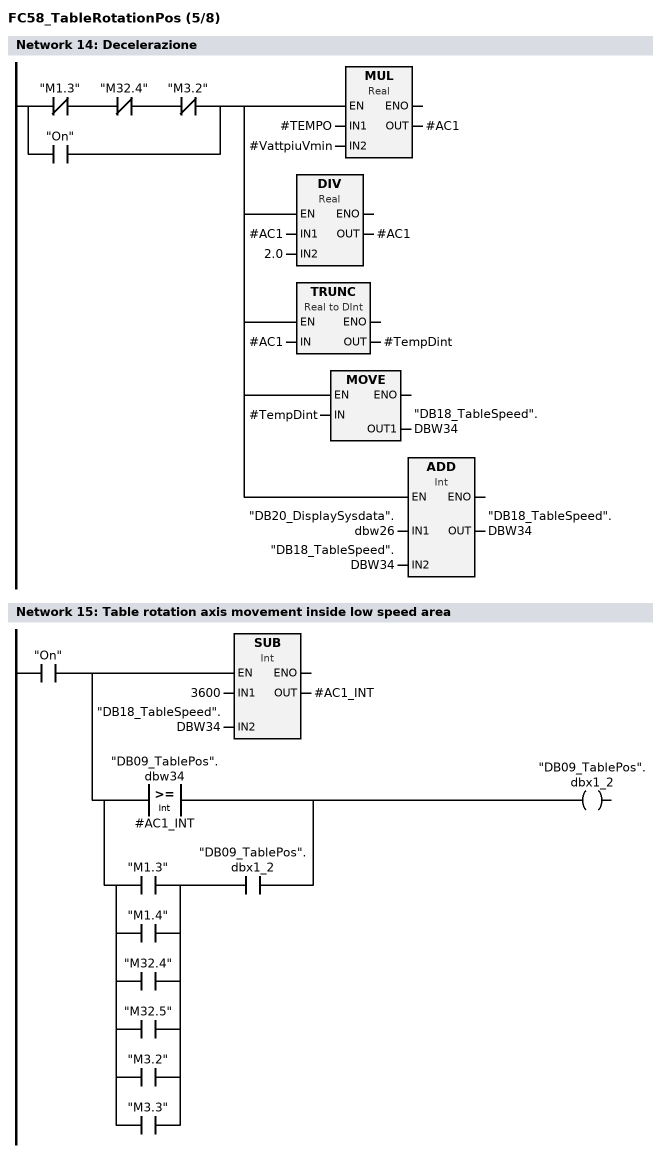
   RUNG wire#powerrail
      I_Contact( "M1.3" )
      I_Contact( "M32.4" )
      I_Contact( "M3.2" )
      wire#w1
      { S7_Templates := "SrcType := Real"; S7_GenerateENO := "TRUE" } Mul(in1 := #TEMPO, in2 := #VattpiuVmin, out => #AC1)
   END_RUNG
   RUNG wire#powerrail
      Contact( "On" )
   END_RUNG wire#w1
   RUNG wire#w1
      { S7_Templates := "SrcType := Real"; S7_GenerateENO := "TRUE" } Div(in1 := #AC1, in2 := 2.0, out => #AC1)
   END_RUNG
   RUNG wire#w1
      { S7_Templates := "[SrcType := Real, DestType := DInt]"; S7_GenerateENO := "TRUE" } Trunc(in := #AC1, out => #TempDint)
   END_RUNG
   RUNG wire#w1
      { S7_GenerateENO := "TRUE" } Move(in := #TempDint, out1 => "DB18_TableSpeed".DBW34)
   END_RUNG
   RUNG wire#w1
      { S7_Templates := "SrcType := Int"; S7_GenerateENO := "TRUE" } Add(in1 := "DB20_DisplaySysdata".dbw26, in2 := "DB18_TableSpeed".DBW34, out => "DB18_TableSpeed".DBW34)
   END_RUNG
   // the same network as SCL:
   IF (NOT "M1.3" AND NOT "M32.4" AND NOT "M3.2") OR "On" THEN
       #AC1 := #TEMPO * #VattpiuVmin;
       #AC1 := #AC1 / 2.0;
       #TempDint := TRUNC(#AC1);
       "DB18_TableSpeed".DBW34 := #TempDint;
       "DB18_TableSpeed".DBW34 := "DB20_DisplaySysdata".dbw26 + "DB18_TableSpeed".DBW34;
   END_IF;
END_REGION

REGION Network 15: Table rotation axis movement inside low speed area
   RUNG wire#powerrail
      Contact( "On" )
      wire#w1
      { S7_Templates := "SrcType := Int"; S7_GenerateENO := "TRUE" } Sub(in1 := 3600, in2 := "DB18_TableSpeed".DBW34, out => #AC1_INT)
   END_RUNG
   RUNG wire#w1
      { S7_Templates := "SrcType := Int" } GE_Contact(in1 := "DB09_TablePos".dbw34, in2 := #AC1_INT)
      wire#w2
      Coil( "DB09_TablePos".dbx1_2 )
   END_RUNG
   RUNG wire#w1
      Contact( "M1.3" )
      wire#w3
      Contact( "DB09_TablePos".dbx1_2 )
   END_RUNG wire#w2
   RUNG wire#w1
      Contact( "M1.4" )
   END_RUNG wire#w3
   RUNG wire#w1
      Contact( "M32.4" )
   END_RUNG wire#w3
   RUNG wire#w1
      Contact( "M32.5" )
   END_RUNG wire#w3
   RUNG wire#w1
      Contact( "M3.2" )
   END_RUNG wire#w3
   RUNG wire#w1
      Contact( "M3.3" )
   END_RUNG wire#w3
   // the same network as SCL:
   IF "On" THEN #AC1_INT := 3600 - "DB18_TableSpeed".DBW34; END_IF;
   "DB09_TablePos".dbx1_2 := "On" AND (("DB09_TablePos".dbw34 >= #AC1_INT) OR (("M1.3" OR "M1.4" OR "M32.4" OR "M32.5" OR "M3.2" OR "M3.3") AND "DB09_TablePos".dbx1_2));
END_REGION

REGION Network 16: Table rotation position loading/Unloading
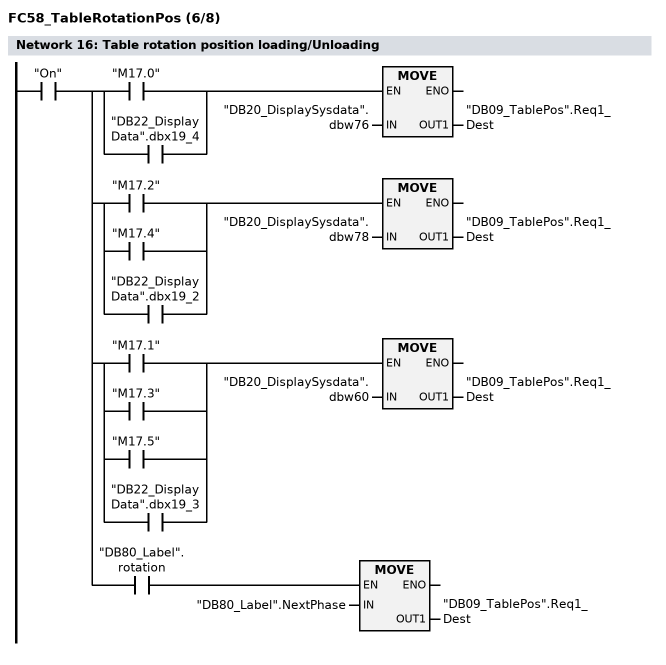
   RUNG wire#powerrail
      Contact( "On" )
      wire#w1
      Contact( "M17.0" )
      wire#w2
      { S7_GenerateENO := "TRUE" } Move(in := "DB20_DisplaySysdata".dbw76, out1 => "DB09_TablePos".Req1_Dest)
   END_RUNG
   RUNG wire#w1
      Contact( "DB22_DisplayData".dbx19_4 )
   END_RUNG wire#w2
   RUNG wire#w1
      Contact( "M17.2" )
      wire#w3
      { S7_GenerateENO := "TRUE" } Move(in := "DB20_DisplaySysdata".dbw78, out1 => "DB09_TablePos".Req1_Dest)
   END_RUNG
   RUNG wire#w1
      Contact( "M17.4" )
   END_RUNG wire#w3
   RUNG wire#w1
      Contact( "DB22_DisplayData".dbx19_2 )
   END_RUNG wire#w3
   RUNG wire#w1
      Contact( "M17.1" )
      wire#w4
      { S7_GenerateENO := "TRUE" } Move(in := "DB20_DisplaySysdata".dbw60, out1 => "DB09_TablePos".Req1_Dest)
   END_RUNG
   RUNG wire#w1
      Contact( "M17.3" )
   END_RUNG wire#w4
   RUNG wire#w1
      Contact( "M17.5" )
   END_RUNG wire#w4
   RUNG wire#w1
      Contact( "DB22_DisplayData".dbx19_3 )
   END_RUNG wire#w4
   RUNG wire#w1
      Contact( "DB80_Label".rotation )
      { S7_GenerateENO := "TRUE" } Move(in := "DB80_Label".NextPhase, out1 => "DB09_TablePos".Req1_Dest)
   END_RUNG
   // the same network as SCL:
   IF "On" AND ("M17.0" OR "DB22_DisplayData".dbx19_4) THEN
       "DB09_TablePos".Req1_Dest := "DB20_DisplaySysdata".dbw76;
   END_IF;
   IF "On" AND ("M17.2" OR "M17.4" OR "DB22_DisplayData".dbx19_2) THEN
       "DB09_TablePos".Req1_Dest := "DB20_DisplaySysdata".dbw78;
   END_IF;
   IF "On" AND ("M17.1" OR "M17.3" OR "M17.5" OR "DB22_DisplayData".dbx19_3) THEN
       "DB09_TablePos".Req1_Dest := "DB20_DisplaySysdata".dbw60;
   END_IF;
   IF "On" AND "DB80_Label".rotation THEN "DB09_TablePos".Req1_Dest := "DB80_Label".NextPhase; END_IF;
END_REGION

REGION Network 17
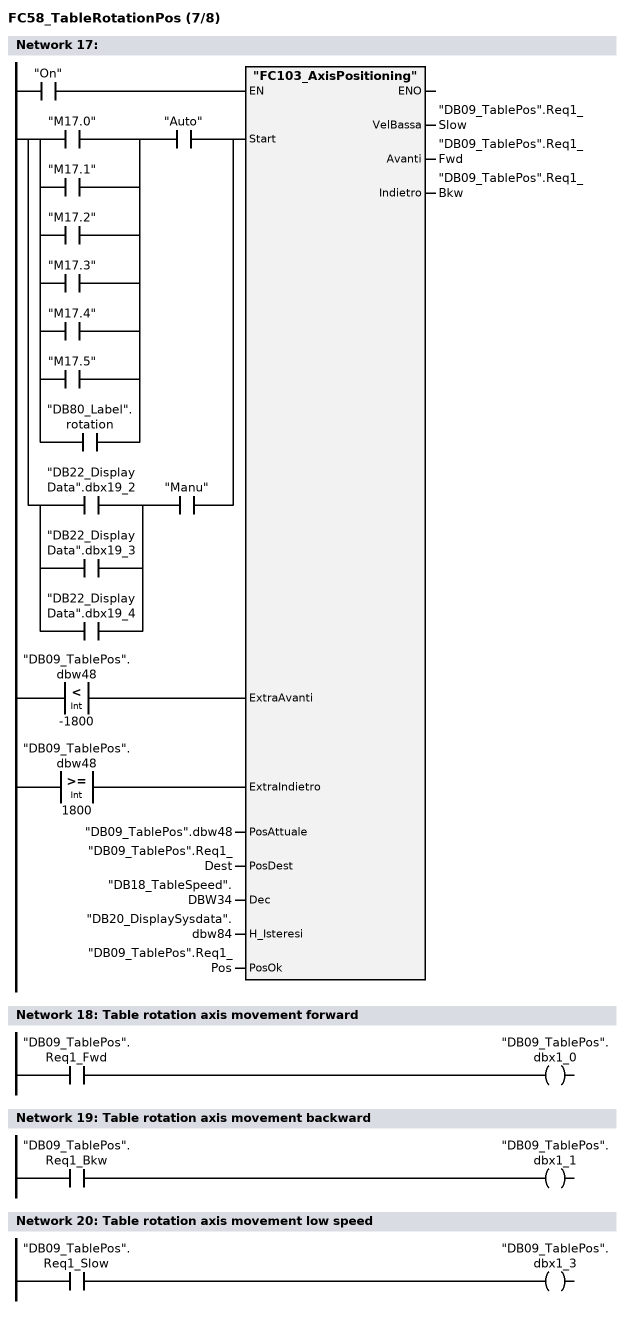
   RUNG wire#powerrail
      Contact( "On" )
      "FC103_AxisPositioning"(Start := wire#w3, ExtraAvanti := wire#w4, ExtraIndietro := wire#w5, PosAttuale := "DB09_TablePos".dbw48, PosDest := "DB09_TablePos".Req1_Dest, Dec := "DB18_TableSpeed".DBW34, H_Isteresi := "DB20_DisplaySysdata".dbw84, PosOk := "DB09_TablePos".Req1_Pos, VelBassa => "DB09_TablePos".Req1_Slow, Avanti => "DB09_TablePos".Req1_Fwd, Indietro => "DB09_TablePos".Req1_Bkw)
   END_RUNG
   RUNG wire#powerrail
      Contact( "M17.0" )
      wire#w1
      Contact( "Auto" )
   END_RUNG wire#w3
   RUNG wire#powerrail
      Contact( "M17.1" )
   END_RUNG wire#w1
   RUNG wire#powerrail
      Contact( "M17.2" )
   END_RUNG wire#w1
   RUNG wire#powerrail
      Contact( "M17.3" )
   END_RUNG wire#w1
   RUNG wire#powerrail
      Contact( "M17.4" )
   END_RUNG wire#w1
   RUNG wire#powerrail
      Contact( "M17.5" )
   END_RUNG wire#w1
   RUNG wire#powerrail
      Contact( "DB80_Label".rotation )
   END_RUNG wire#w1
   RUNG wire#powerrail
      Contact( "DB22_DisplayData".dbx19_2 )
      wire#w2
      Contact( "Manu" )
   END_RUNG wire#w3
   RUNG wire#powerrail
      Contact( "DB22_DisplayData".dbx19_3 )
   END_RUNG wire#w2
   RUNG wire#powerrail
      Contact( "DB22_DisplayData".dbx19_4 )
   END_RUNG wire#w2
   RUNG wire#powerrail
      { S7_Templates := "SrcType := Int" } LT_Contact(in1 := "DB09_TablePos".dbw48, in2 := -1800)
   END_RUNG wire#w4
   RUNG wire#powerrail
      { S7_Templates := "SrcType := Int" } GE_Contact(in1 := "DB09_TablePos".dbw48, in2 := 1800)
   END_RUNG wire#w5
   // the same network as SCL:
   IF "On" THEN
       "FC103_AxisPositioning"(Start := (("M17.0" OR "M17.1" OR "M17.2" OR "M17.3" OR "M17.4" OR "M17.5" OR "DB80_Label".rotation) AND "Auto") OR (("DB22_DisplayData".dbx19_2 OR "DB22_DisplayData".dbx19_3 OR "DB22_DisplayData".dbx19_4) AND "Manu"),
                               ExtraAvanti := "DB09_TablePos".dbw48 < (-1800),
                               ExtraIndietro := "DB09_TablePos".dbw48 >= 1800,
                               PosAttuale := "DB09_TablePos".dbw48,
                               PosDest := "DB09_TablePos".Req1_Dest,
                               Dec := "DB18_TableSpeed".DBW34,
                               H_Isteresi := "DB20_DisplaySysdata".dbw84,
                               PosOk := "DB09_TablePos".Req1_Pos,
                               VelBassa => "DB09_TablePos".Req1_Slow,
                               Avanti => "DB09_TablePos".Req1_Fwd,
                               Indietro => "DB09_TablePos".Req1_Bkw);
   END_IF;
END_REGION

REGION Network 18: Table rotation axis movement forward
   RUNG wire#powerrail
      Contact( "DB09_TablePos".Req1_Fwd )
      Coil( "DB09_TablePos".dbx1_0 )
   END_RUNG
   // the same network as SCL:
   "DB09_TablePos".dbx1_0 := "DB09_TablePos".Req1_Fwd;
END_REGION

REGION Network 19: Table rotation axis movement backward
   RUNG wire#powerrail
      Contact( "DB09_TablePos".Req1_Bkw )
      Coil( "DB09_TablePos".dbx1_1 )
   END_RUNG
   // the same network as SCL:
   "DB09_TablePos".dbx1_1 := "DB09_TablePos".Req1_Bkw;
END_REGION

REGION Network 20: Table rotation axis movement low speed
   RUNG wire#powerrail
      Contact( "DB09_TablePos".Req1_Slow )
      Coil( "DB09_TablePos".dbx1_3 )
   END_RUNG
   // the same network as SCL:
   "DB09_TablePos".dbx1_3 := "DB09_TablePos".Req1_Slow;
END_REGION

REGION Network 21: TABLE ENCODER CHECK
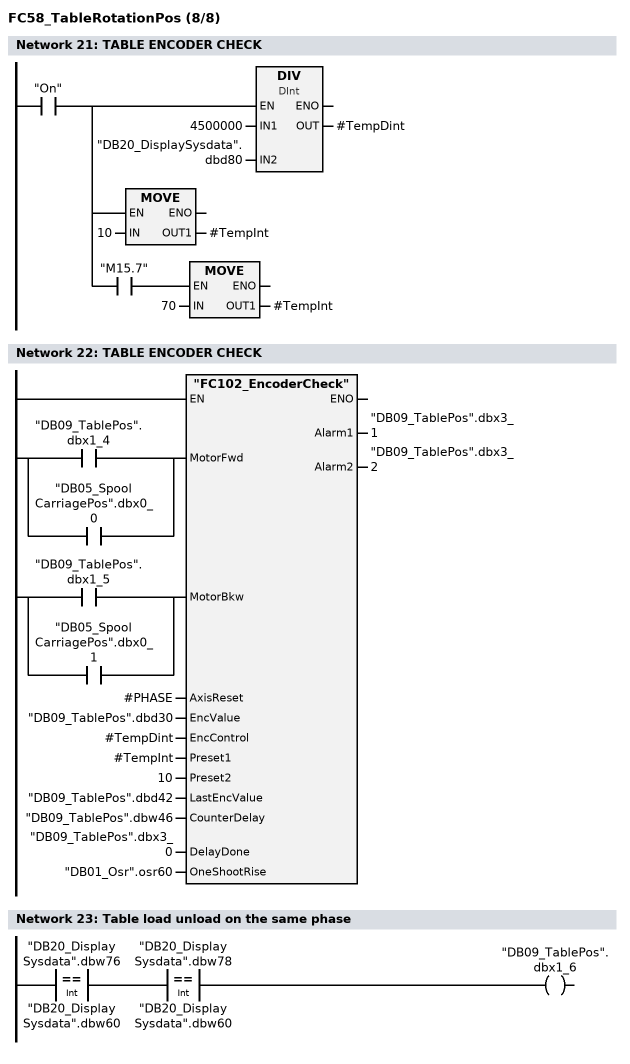
   RUNG wire#powerrail
      Contact( "On" )
      wire#w1
      { S7_Templates := "SrcType := DInt"; S7_GenerateENO := "TRUE" } Div(in1 := 4500000, in2 := "DB20_DisplaySysdata".dbd80, out => #TempDint)
   END_RUNG
   RUNG wire#w1
      { S7_GenerateENO := "TRUE" } Move(in := 10, out1 => #TempInt)
   END_RUNG
   RUNG wire#w1
      Contact( "M15.7" )
      { S7_GenerateENO := "TRUE" } Move(in := 70, out1 => #TempInt)
   END_RUNG
   // the same network as SCL:
   IF "On" THEN
       #TempDint := 4500000 / "DB20_DisplaySysdata".dbd80;
       #TempInt := 10;
   END_IF;
   IF "On" AND "M15.7" THEN #TempInt := 70; END_IF;
END_REGION

REGION Network 22: TABLE ENCODER CHECK
   RUNG wire#powerrail
      "FC102_EncoderCheck"(MotorFwd := wire#w1, MotorBkw := wire#w2, AxisReset := #PHASE, EncValue := "DB09_TablePos".dbd30, EncControl := #TempDint, Preset1 := #TempInt, Preset2 := 10, LastEncValue := "DB09_TablePos".dbd42, CounterDelay := "DB09_TablePos".dbw46, DelayDone := "DB09_TablePos".dbx3_0, OneShootRise := "DB01_Osr".osr60, Alarm1 => "DB09_TablePos".dbx3_1, Alarm2 => "DB09_TablePos".dbx3_2)
   END_RUNG
   RUNG wire#powerrail
      Contact( "DB09_TablePos".dbx1_4 )
   END_RUNG wire#w1
   RUNG wire#powerrail
      Contact( "DB05_SpoolCarriagePos".dbx0_0 )
   END_RUNG wire#w1
   RUNG wire#powerrail
      Contact( "DB09_TablePos".dbx1_5 )
   END_RUNG wire#w2
   RUNG wire#powerrail
      Contact( "DB05_SpoolCarriagePos".dbx0_1 )
   END_RUNG wire#w2
   // the same network as SCL:
   "FC102_EncoderCheck"(MotorFwd := "DB09_TablePos".dbx1_4 OR "DB05_SpoolCarriagePos".dbx0_0,
                        MotorBkw := "DB09_TablePos".dbx1_5 OR "DB05_SpoolCarriagePos".dbx0_1,
                        AxisReset := #PHASE,
                        EncValue := "DB09_TablePos".dbd30,
                        EncControl := #TempDint,
                        Preset1 := #TempInt,
                        Preset2 := 10,
                        LastEncValue := "DB09_TablePos".dbd42,
                        CounterDelay := "DB09_TablePos".dbw46,
                        DelayDone := "DB09_TablePos".dbx3_0,
                        OneShootRise := "DB01_Osr".osr60,
                        Alarm1 => "DB09_TablePos".dbx3_1,
                        Alarm2 => "DB09_TablePos".dbx3_2);
END_REGION

REGION Network 23: Table load unload on the same phase
   RUNG wire#powerrail
      { S7_Templates := "SrcType := Int" } EQ_Contact(in1 := "DB20_DisplaySysdata".dbw76, in2 := "DB20_DisplaySysdata".dbw60)
      { S7_Templates := "SrcType := Int" } EQ_Contact(in1 := "DB20_DisplaySysdata".dbw78, in2 := "DB20_DisplaySysdata".dbw60)
      Coil( "DB09_TablePos".dbx1_6 )
   END_RUNG
   // the same network as SCL:
   "DB09_TablePos".dbx1_6 := ("DB20_DisplaySysdata".dbw76 = "DB20_DisplaySysdata".dbw60) AND ("DB20_DisplaySysdata".dbw78 = "DB20_DisplaySysdata".dbw60);
END_REGION
END_FUNCTION

FUNCTION "FC62_PreStretchPGSAoutPWM" : Void   // FC62, LAD
{ S7_Optimized_Access := 'FALSE' }
AUTHOR : PaZan
VERSION : 0.1
// stored: AutoNumber false, IsIECCheckEnabled false, SetENOAutomatically false, UDAEnableTagReadback false
BEGIN

REGION Network 1: copy parameter for scale value % prestretch
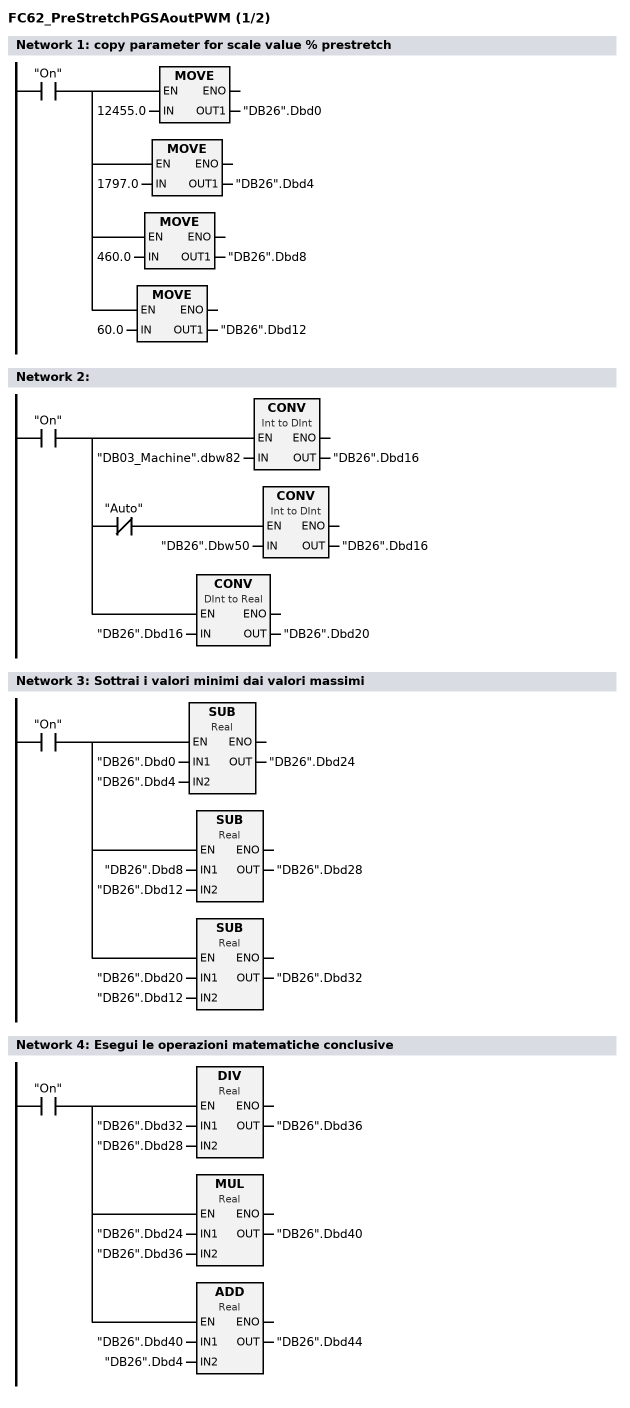
   RUNG wire#powerrail
      Contact( "On" )
      wire#w1
      { S7_GenerateENO := "TRUE" } Move(in := 12455.0, out1 => "DB26".Dbd0)
   END_RUNG
   RUNG wire#w1
      { S7_GenerateENO := "TRUE" } Move(in := 1797.0, out1 => "DB26".Dbd4)
   END_RUNG
   RUNG wire#w1
      { S7_GenerateENO := "TRUE" } Move(in := 460.0, out1 => "DB26".Dbd8)
   END_RUNG
   RUNG wire#w1
      { S7_GenerateENO := "TRUE" } Move(in := 60.0, out1 => "DB26".Dbd12)
   END_RUNG
   // the same network as SCL:
   IF "On" THEN
       "DB26".Dbd0 := 12455.0;
       "DB26".Dbd4 := 1797.0;
       "DB26".Dbd8 := 460.0;
       "DB26".Dbd12 := 60.0;
   END_IF;
END_REGION

REGION Network 2
   RUNG wire#powerrail
      Contact( "On" )
      wire#w1
      { S7_Templates := "[SrcType := Int, DestType := DInt]"; S7_GenerateENO := "TRUE" } Convert(in := "DB03_Machine".dbw82, out => "DB26".Dbd16)
   END_RUNG
   RUNG wire#w1
      I_Contact( "Auto" )
      { S7_Templates := "[SrcType := Int, DestType := DInt]"; S7_GenerateENO := "TRUE" } Convert(in := "DB26".Dbw50, out => "DB26".Dbd16)
   END_RUNG
   RUNG wire#w1
      { S7_Templates := "[SrcType := DInt, DestType := Real]"; S7_GenerateENO := "TRUE" } Convert(in := "DB26".Dbd16, out => "DB26".Dbd20)
   END_RUNG
   // the same network as SCL:
   IF "On" THEN "DB26".Dbd16 := INT_TO_DINT("DB03_Machine".dbw82); END_IF;
   IF "On" AND NOT "Auto" THEN "DB26".Dbd16 := INT_TO_DINT("DB26".Dbw50); END_IF;
   IF "On" THEN "DB26".Dbd20 := DINT_TO_REAL("DB26".Dbd16); END_IF;
END_REGION

REGION Network 3: Sottrai i valori minimi dai valori massimi
   RUNG wire#powerrail
      Contact( "On" )
      wire#w1
      { S7_Templates := "SrcType := Real"; S7_GenerateENO := "TRUE" } Sub(in1 := "DB26".Dbd0, in2 := "DB26".Dbd4, out => "DB26".Dbd24)
   END_RUNG
   RUNG wire#w1
      { S7_Templates := "SrcType := Real"; S7_GenerateENO := "TRUE" } Sub(in1 := "DB26".Dbd8, in2 := "DB26".Dbd12, out => "DB26".Dbd28)
   END_RUNG
   RUNG wire#w1
      { S7_Templates := "SrcType := Real"; S7_GenerateENO := "TRUE" } Sub(in1 := "DB26".Dbd20, in2 := "DB26".Dbd12, out => "DB26".Dbd32)
   END_RUNG
   // the same network as SCL:
   IF "On" THEN
       "DB26".Dbd24 := "DB26".Dbd0 - "DB26".Dbd4;
       "DB26".Dbd28 := "DB26".Dbd8 - "DB26".Dbd12;
       "DB26".Dbd32 := "DB26".Dbd20 - "DB26".Dbd12;
   END_IF;
END_REGION

REGION Network 4: Esegui le operazioni matematiche conclusive
   RUNG wire#powerrail
      Contact( "On" )
      wire#w1
      { S7_Templates := "SrcType := Real"; S7_GenerateENO := "TRUE" } Div(in1 := "DB26".Dbd32, in2 := "DB26".Dbd28, out => "DB26".Dbd36)
   END_RUNG
   RUNG wire#w1
      { S7_Templates := "SrcType := Real"; S7_GenerateENO := "TRUE" } Mul(in1 := "DB26".Dbd24, in2 := "DB26".Dbd36, out => "DB26".Dbd40)
   END_RUNG
   RUNG wire#w1
      { S7_Templates := "SrcType := Real"; S7_GenerateENO := "TRUE" } Add(in1 := "DB26".Dbd40, in2 := "DB26".Dbd4, out => "DB26".Dbd44)
   END_RUNG
   // the same network as SCL:
   IF "On" THEN
       "DB26".Dbd36 := "DB26".Dbd32 / "DB26".Dbd28;
       "DB26".Dbd40 := "DB26".Dbd24 * "DB26".Dbd36;
       "DB26".Dbd44 := "DB26".Dbd40 + "DB26".Dbd4;
   END_IF;
END_REGION

REGION Network 5: Trunc and copy value for pre-stretch in analogic out
   // PAW128
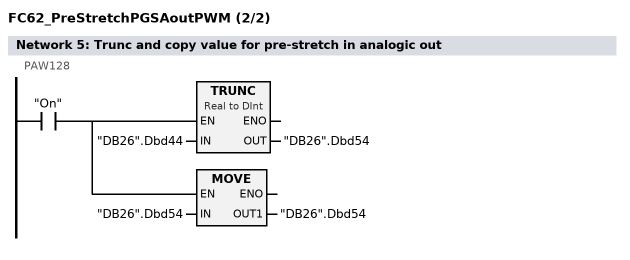
   RUNG wire#powerrail
      Contact( "On" )
      wire#w1
      { S7_Templates := "[SrcType := Real, DestType := DInt]"; S7_GenerateENO := "TRUE" } Trunc(in := "DB26".Dbd44, out => "DB26".Dbd54)
   END_RUNG
   RUNG wire#w1
      { S7_GenerateENO := "TRUE" } Move(in := "DB26".Dbd54, out1 => "DB26".Dbd54)
   END_RUNG
   // the same network as SCL:
   IF "On" THEN
       "DB26".Dbd54 := TRUNC("DB26".Dbd44);
       "DB26".Dbd54 := "DB26".Dbd54;
   END_IF;
END_REGION
END_FUNCTION

FUNCTION "FC71_Conveyor_0_IN_0_OUT" : Void   // FC71, LAD
TITLE = Conveyor_0_IN_0_OUT
{ S7_Optimized_Access := 'FALSE' }
VERSION : 0.1
// stored: AutoNumber false, IsIECCheckEnabled false, SetENOAutomatically false, UDAEnableTagReadback false
BEGIN

REGION Network 1: Conveyor manual movement
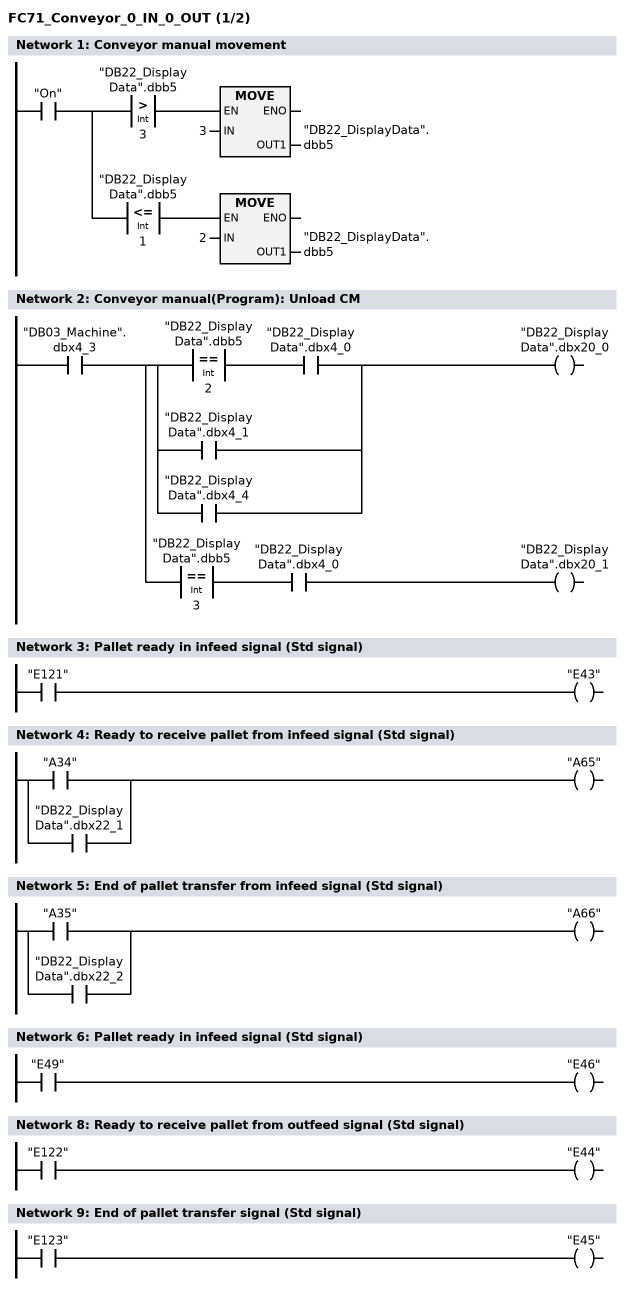
   RUNG wire#powerrail
      Contact( "On" )
      wire#w1
      { S7_Templates := "SrcType := Int" } GT_Contact(in1 := "DB22_DisplayData".dbb5, in2 := 3)
      { S7_GenerateENO := "TRUE" } Move(in := 3, out1 => "DB22_DisplayData".dbb5)
   END_RUNG
   RUNG wire#w1
      { S7_Templates := "SrcType := Int" } LE_Contact(in1 := "DB22_DisplayData".dbb5, in2 := 1)
      { S7_GenerateENO := "TRUE" } Move(in := 2, out1 => "DB22_DisplayData".dbb5)
   END_RUNG
   // the same network as SCL:
   IF "On" AND ("DB22_DisplayData".dbb5 > 3) THEN "DB22_DisplayData".dbb5 := 3; END_IF;
   IF "On" AND ("DB22_DisplayData".dbb5 <= 1) THEN "DB22_DisplayData".dbb5 := 2; END_IF;
END_REGION

REGION Network 2: Conveyor manual(Program): Unload CM
   RUNG wire#powerrail
      Contact( "DB03_Machine".dbx4_3 )
      wire#w1
      { S7_Templates := "SrcType := Int" } EQ_Contact(in1 := "DB22_DisplayData".dbb5, in2 := 2)
      Contact( "DB22_DisplayData".dbx4_0 )
      wire#w2
      Coil( "DB22_DisplayData".dbx20_0 )
   END_RUNG
   RUNG wire#w1
      Contact( "DB22_DisplayData".dbx4_1 )
   END_RUNG wire#w2
   RUNG wire#w1
      Contact( "DB22_DisplayData".dbx4_4 )
   END_RUNG wire#w2
   RUNG wire#w1
      { S7_Templates := "SrcType := Int" } EQ_Contact(in1 := "DB22_DisplayData".dbb5, in2 := 3)
      Contact( "DB22_DisplayData".dbx4_0 )
      Coil( "DB22_DisplayData".dbx20_1 )
   END_RUNG
   // the same network as SCL:
   "DB22_DisplayData".dbx20_0 := "DB03_Machine".dbx4_3 AND ((("DB22_DisplayData".dbb5 = 2) AND "DB22_DisplayData".dbx4_0) OR "DB22_DisplayData".dbx4_1 OR "DB22_DisplayData".dbx4_4);
   "DB22_DisplayData".dbx20_1 := "DB03_Machine".dbx4_3 AND ("DB22_DisplayData".dbb5 = 3) AND "DB22_DisplayData".dbx4_0;
END_REGION

REGION Network 3: Pallet ready in infeed signal (Std signal)
   RUNG wire#powerrail
      Contact( "E121" )
      Coil( "E43" )
   END_RUNG
   // the same network as SCL:
   "E43" := "E121";
END_REGION

REGION Network 4: Ready to receive pallet from infeed signal (Std signal)
   RUNG wire#powerrail
      Contact( "A34" )
      wire#w1
      Coil( "A65" )
   END_RUNG
   RUNG wire#powerrail
      Contact( "DB22_DisplayData".dbx22_1 )
   END_RUNG wire#w1
   // the same network as SCL:
   "A65" := "A34" OR "DB22_DisplayData".dbx22_1;
END_REGION

REGION Network 5: End of pallet transfer from infeed signal (Std signal)
   RUNG wire#powerrail
      Contact( "A35" )
      wire#w1
      Coil( "A66" )
   END_RUNG
   RUNG wire#powerrail
      Contact( "DB22_DisplayData".dbx22_2 )
   END_RUNG wire#w1
   // the same network as SCL:
   "A66" := "A35" OR "DB22_DisplayData".dbx22_2;
END_REGION

REGION Network 6: Pallet ready in infeed signal (Std signal)
   RUNG wire#powerrail
      Contact( "E49" )
      Coil( "E46" )
   END_RUNG
   // the same network as SCL:
   "E46" := "E49";
END_REGION

REGION Network 7: >>>>> OUTFEED CONVEYOR <<<<<<
END_REGION

REGION Network 8: Ready to receive pallet from outfeed signal (Std signal)
   RUNG wire#powerrail
      Contact( "E122" )
      Coil( "E44" )
   END_RUNG
   // the same network as SCL:
   "E44" := "E122";
END_REGION

REGION Network 9: End of pallet transfer signal (Std signal)
   RUNG wire#powerrail
      Contact( "E123" )
      Coil( "E45" )
   END_RUNG
   // the same network as SCL:
   "E45" := "E123";
END_REGION

REGION Network 10: Pallet ready for outfeed signal (Std signal)
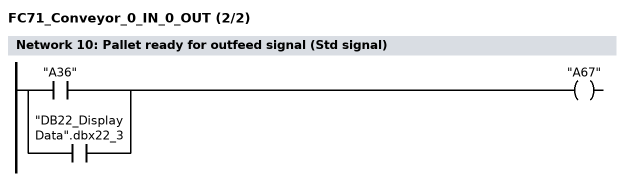
   RUNG wire#powerrail
      Contact( "A36" )
      wire#w1
      Coil( "A67" )
   END_RUNG
   RUNG wire#powerrail
      Contact( "DB22_DisplayData".dbx22_3 )
   END_RUNG wire#w1
   // the same network as SCL:
   "A67" := "A36" OR "DB22_DisplayData".dbx22_3;
END_REGION
END_FUNCTION

FUNCTION "FC72_Conveyor_0_IN_1_OUT" : Void   // FC72, LAD
TITLE = Conveyor_0_IN_1_OUT
{ S7_Optimized_Access := 'FALSE' }
VERSION : 0.1
// stored: AutoNumber false, IsIECCheckEnabled false, SetENOAutomatically false, UDAEnableTagReadback false
   VAR_TEMP   // added for the SCL form of the ladder/FBD networks
      _w1 : Bool;
   END_VAR
BEGIN

REGION Network 1: Conveyor manual movement
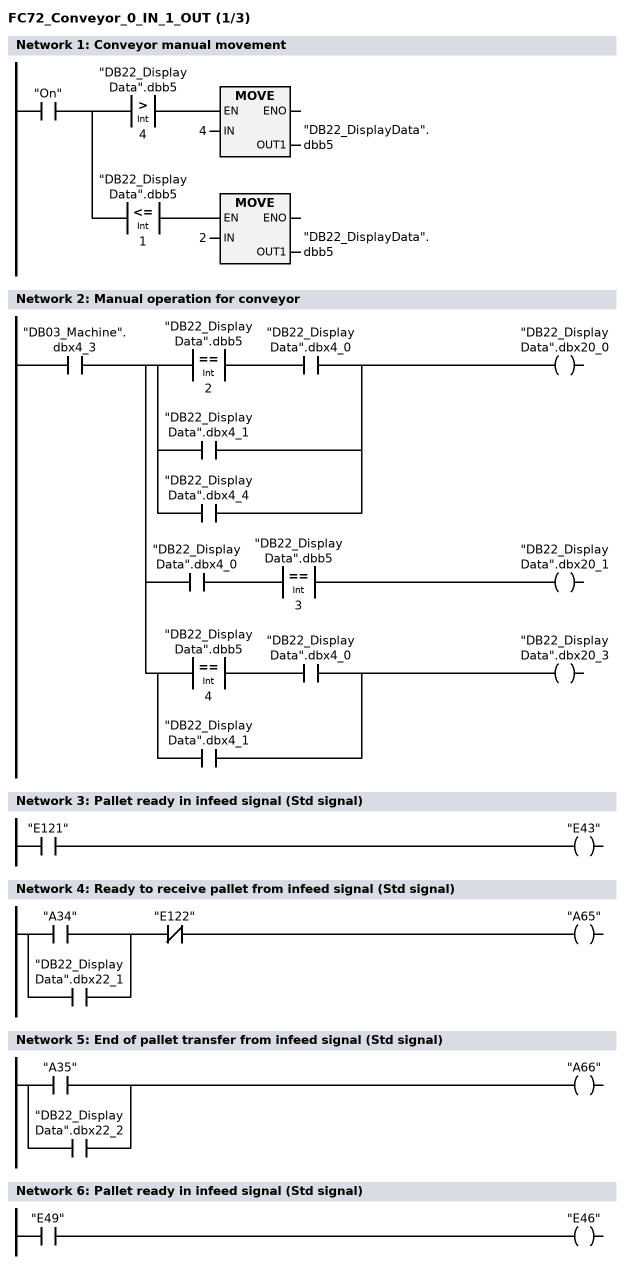
   RUNG wire#powerrail
      Contact( "On" )
      wire#w1
      { S7_Templates := "SrcType := Int" } GT_Contact(in1 := "DB22_DisplayData".dbb5, in2 := 4)
      { S7_GenerateENO := "TRUE" } Move(in := 4, out1 => "DB22_DisplayData".dbb5)
   END_RUNG
   RUNG wire#w1
      { S7_Templates := "SrcType := Int" } LE_Contact(in1 := "DB22_DisplayData".dbb5, in2 := 1)
      { S7_GenerateENO := "TRUE" } Move(in := 2, out1 => "DB22_DisplayData".dbb5)
   END_RUNG
   // the same network as SCL:
   IF "On" AND ("DB22_DisplayData".dbb5 > 4) THEN "DB22_DisplayData".dbb5 := 4; END_IF;
   IF "On" AND ("DB22_DisplayData".dbb5 <= 1) THEN "DB22_DisplayData".dbb5 := 2; END_IF;
END_REGION

REGION Network 2: Manual operation for conveyor
   RUNG wire#powerrail
      Contact( "DB03_Machine".dbx4_3 )
      wire#w1
      { S7_Templates := "SrcType := Int" } EQ_Contact(in1 := "DB22_DisplayData".dbb5, in2 := 2)
      Contact( "DB22_DisplayData".dbx4_0 )
      wire#w2
      Coil( "DB22_DisplayData".dbx20_0 )
   END_RUNG
   RUNG wire#w1
      Contact( "DB22_DisplayData".dbx4_1 )
   END_RUNG wire#w2
   RUNG wire#w1
      Contact( "DB22_DisplayData".dbx4_4 )
   END_RUNG wire#w2
   RUNG wire#w1
      Contact( "DB22_DisplayData".dbx4_0 )
      { S7_Templates := "SrcType := Int" } EQ_Contact(in1 := "DB22_DisplayData".dbb5, in2 := 3)
      Coil( "DB22_DisplayData".dbx20_1 )
   END_RUNG
   RUNG wire#w1
      { S7_Templates := "SrcType := Int" } EQ_Contact(in1 := "DB22_DisplayData".dbb5, in2 := 4)
      Contact( "DB22_DisplayData".dbx4_0 )
      wire#w3
      Coil( "DB22_DisplayData".dbx20_3 )
   END_RUNG
   RUNG wire#w1
      Contact( "DB22_DisplayData".dbx4_1 )
   END_RUNG wire#w3
   // the same network as SCL:
   "DB22_DisplayData".dbx20_0 := "DB03_Machine".dbx4_3 AND ((("DB22_DisplayData".dbb5 = 2) AND "DB22_DisplayData".dbx4_0) OR "DB22_DisplayData".dbx4_1 OR "DB22_DisplayData".dbx4_4);
   "DB22_DisplayData".dbx20_1 := "DB03_Machine".dbx4_3 AND "DB22_DisplayData".dbx4_0 AND ("DB22_DisplayData".dbb5 = 3);
   "DB22_DisplayData".dbx20_3 := "DB03_Machine".dbx4_3 AND ((("DB22_DisplayData".dbb5 = 4) AND "DB22_DisplayData".dbx4_0) OR "DB22_DisplayData".dbx4_1);
END_REGION

REGION Network 3: Pallet ready in infeed signal (Std signal)
   RUNG wire#powerrail
      Contact( "E121" )
      Coil( "E43" )
   END_RUNG
   // the same network as SCL:
   "E43" := "E121";
END_REGION

REGION Network 4: Ready to receive pallet from infeed signal (Std signal)
   RUNG wire#powerrail
      Contact( "A34" )
      wire#w1
      I_Contact( "E122" )
      Coil( "A65" )
   END_RUNG
   RUNG wire#powerrail
      Contact( "DB22_DisplayData".dbx22_1 )
   END_RUNG wire#w1
   // the same network as SCL:
   "A65" := ("A34" OR "DB22_DisplayData".dbx22_1) AND NOT "E122";
END_REGION

REGION Network 5: End of pallet transfer from infeed signal (Std signal)
   RUNG wire#powerrail
      Contact( "A35" )
      wire#w1
      Coil( "A66" )
   END_RUNG
   RUNG wire#powerrail
      Contact( "DB22_DisplayData".dbx22_2 )
   END_RUNG wire#w1
   // the same network as SCL:
   "A66" := "A35" OR "DB22_DisplayData".dbx22_2;
END_REGION

REGION Network 6: Pallet ready in infeed signal (Std signal)
   RUNG wire#powerrail
      Contact( "E49" )
      Coil( "E46" )
   END_RUNG
   // the same network as SCL:
   "E46" := "E49";
END_REGION

REGION Network 7: >>>>> OUTFEED CONVEYOR <<<<<<
END_REGION

REGION Network 8: Time for pallet unload with forklift
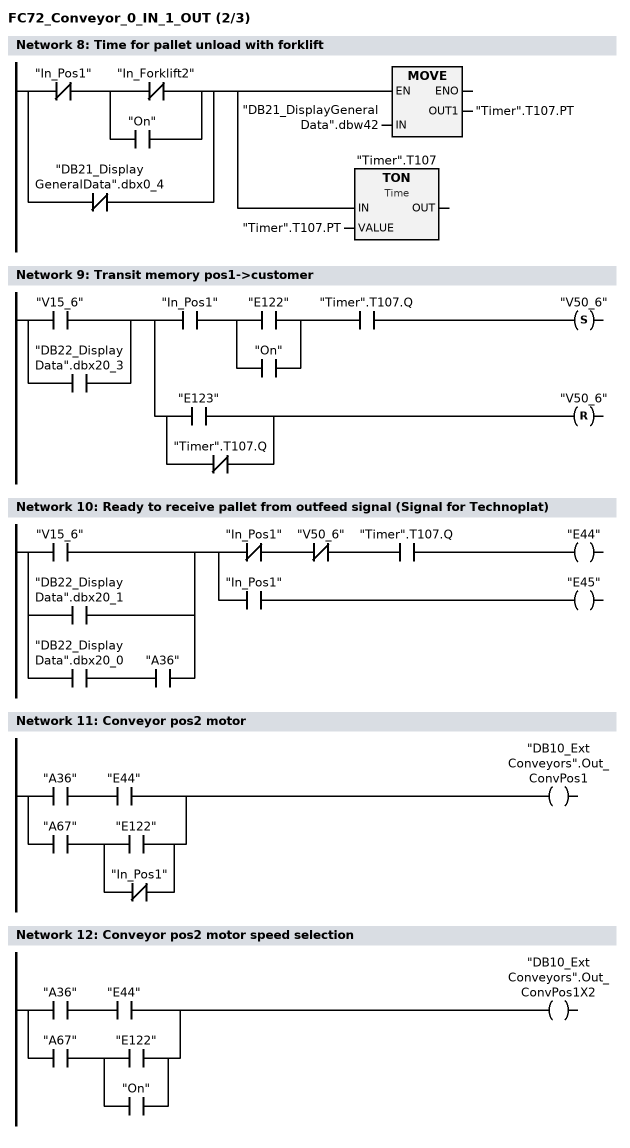
   #_w1 := (NOT "In_Pos1" AND (NOT "In_Forklift2" OR "On")) OR NOT "DB21_DisplayGeneralData".dbx0_4;
   IF #_w1 THEN "Timer".T107.PT := "DB21_DisplayGeneralData".dbw42; END_IF;
   "Timer".T107.TON(IN := #_w1, PT := "Timer".T107.PT);   // TON coil
END_REGION

REGION Network 9: Transit memory pos1->customer
   RUNG wire#powerrail
      Contact( "V15_6" )
      wire#w1
      Contact( "In_Pos1" )
      wire#w2
      Contact( "E122" )
      wire#w3
      Contact( "Timer".T107.Q )
      S_Coil( "V50_6" )
   END_RUNG
   RUNG wire#powerrail
      Contact( "DB22_DisplayData".dbx20_3 )
   END_RUNG wire#w1
   RUNG wire#w2
      Contact( "On" )
   END_RUNG wire#w3
   RUNG wire#w1
      Contact( "E123" )
      wire#w4
      R_Coil( "V50_6" )
   END_RUNG
   RUNG wire#w1
      I_Contact( "Timer".T107.Q )
   END_RUNG wire#w4
   // the same network as SCL:
   #_w1 := "V15_6" OR "DB22_DisplayData".dbx20_3;
   IF #_w1 AND "In_Pos1" AND ("E122" OR "On") AND "Timer".T107.Q THEN "V50_6" := TRUE; END_IF;
   IF #_w1 AND ("E123" OR NOT "Timer".T107.Q) THEN "V50_6" := FALSE; END_IF;
END_REGION

REGION Network 10: Ready to receive pallet from outfeed signal (Signal for Technoplat)
   RUNG wire#powerrail
      Contact( "V15_6" )
      wire#w1
      I_Contact( "In_Pos1" )
      I_Contact( "V50_6" )
      Contact( "Timer".T107.Q )
      Coil( "E44" )
   END_RUNG
   RUNG wire#powerrail
      Contact( "DB22_DisplayData".dbx20_1 )
   END_RUNG wire#w1
   RUNG wire#powerrail
      Contact( "DB22_DisplayData".dbx20_0 )
      Contact( "A36" )
   END_RUNG wire#w1
   RUNG wire#w1
      Contact( "In_Pos1" )
      Coil( "E45" )
   END_RUNG
   // the same network as SCL:
   #_w1 := "V15_6" OR "DB22_DisplayData".dbx20_1 OR ("DB22_DisplayData".dbx20_0 AND "A36");
   "E44" := #_w1 AND NOT "In_Pos1" AND NOT "V50_6" AND "Timer".T107.Q;
   "E45" := #_w1 AND "In_Pos1";
END_REGION

REGION Network 11: Conveyor pos2 motor
   RUNG wire#powerrail
      Contact( "A36" )
      Contact( "E44" )
      wire#w1
      Coil( "DB10_ExtConveyors".Out_ConvPos1 )
   END_RUNG
   RUNG wire#powerrail
      Contact( "A67" )
      wire#w2
      Contact( "E122" )
   END_RUNG wire#w1
   RUNG wire#w2
      I_Contact( "In_Pos1" )
   END_RUNG wire#w1
   // the same network as SCL:
   "DB10_ExtConveyors".Out_ConvPos1 := ("A36" AND "E44") OR ("A67" AND ("E122" OR NOT "In_Pos1"));
END_REGION

REGION Network 12: Conveyor pos2 motor speed selection
   RUNG wire#powerrail
      Contact( "A36" )
      Contact( "E44" )
      wire#w1
      Coil( "DB10_ExtConveyors".Out_ConvPos1X2 )
   END_RUNG
   RUNG wire#powerrail
      Contact( "A67" )
      wire#w2
      Contact( "E122" )
   END_RUNG wire#w1
   RUNG wire#w2
      Contact( "On" )
   END_RUNG wire#w1
   // the same network as SCL:
   "DB10_ExtConveyors".Out_ConvPos1X2 := ("A36" AND "E44") OR ("A67" AND ("E122" OR "On"));
END_REGION

REGION Network 13: Pallet ready in outfeed signal
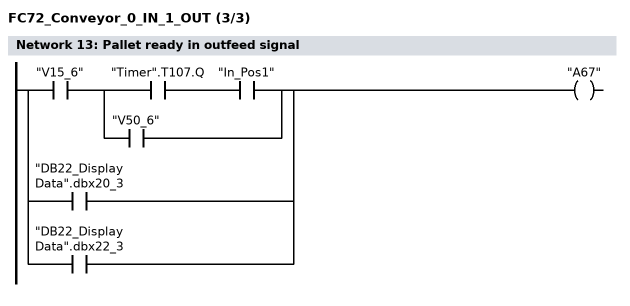
   RUNG wire#powerrail
      Contact( "V15_6" )
      wire#w1
      Contact( "Timer".T107.Q )
      Contact( "In_Pos1" )
      wire#w2
      Coil( "A67" )
   END_RUNG
   RUNG wire#w1
      Contact( "V50_6" )
   END_RUNG wire#w2
   RUNG wire#powerrail
      Contact( "DB22_DisplayData".dbx20_3 )
   END_RUNG wire#w2
   RUNG wire#powerrail
      Contact( "DB22_DisplayData".dbx22_3 )
   END_RUNG wire#w2
   // the same network as SCL:
   "A67" := ("V15_6" AND (("Timer".T107.Q AND "In_Pos1") OR "V50_6")) OR "DB22_DisplayData".dbx20_3 OR "DB22_DisplayData".dbx22_3;
END_REGION
END_FUNCTION

FUNCTION "FC80_Label" : Void   // FC80, LAD
TITLE = Label device
{ S7_Optimized_Access := 'FALSE' }
VERSION : 0.1
// stored: AutoNumber false, IsIECCheckEnabled false, SetENOAutomatically false, UDAEnableTagReadback false
BEGIN

REGION Network 1: Label arm in home position for pallet transit
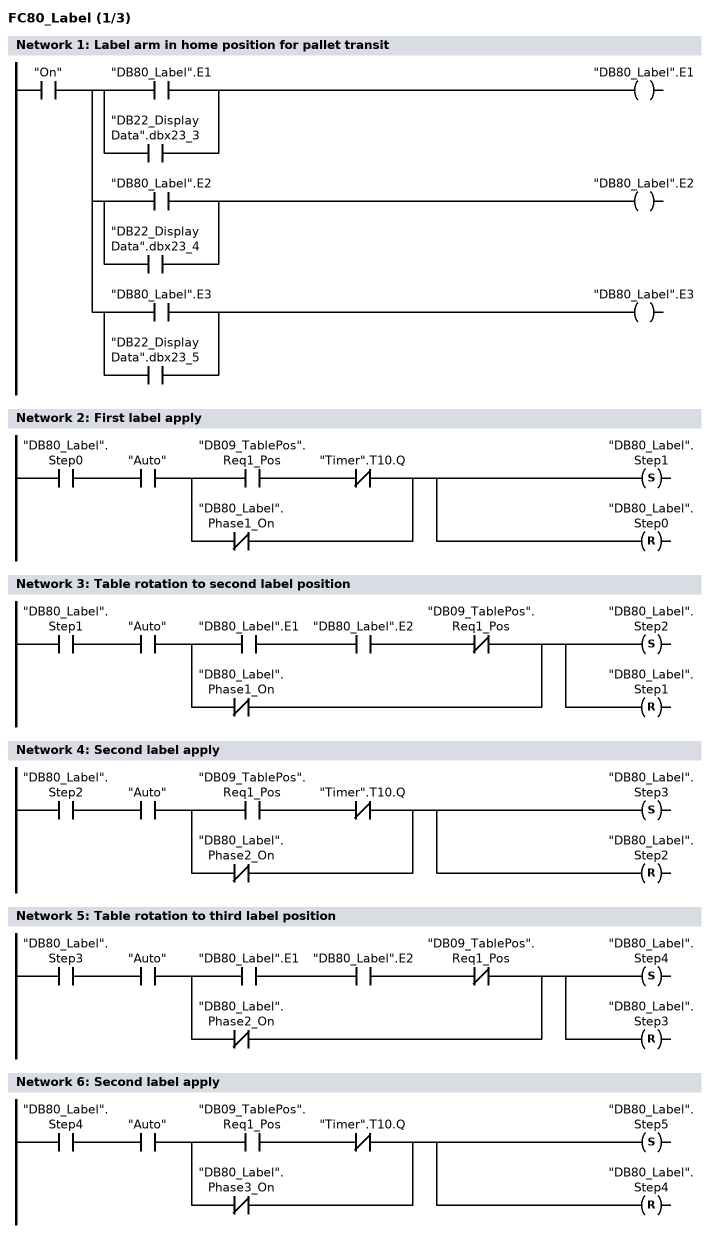
   RUNG wire#powerrail
      Contact( "On" )
      wire#w1
      Contact( "DB80_Label".E1 )
      wire#w2
      Coil( "DB80_Label".E1 )
   END_RUNG
   RUNG wire#w1
      Contact( "DB22_DisplayData".dbx23_3 )
   END_RUNG wire#w2
   RUNG wire#w1
      Contact( "DB80_Label".E2 )
      wire#w3
      Coil( "DB80_Label".E2 )
   END_RUNG
   RUNG wire#w1
      Contact( "DB22_DisplayData".dbx23_4 )
   END_RUNG wire#w3
   RUNG wire#w1
      Contact( "DB80_Label".E3 )
      wire#w4
      Coil( "DB80_Label".E3 )
   END_RUNG
   RUNG wire#w1
      Contact( "DB22_DisplayData".dbx23_5 )
   END_RUNG wire#w4
   // the same network as SCL:
   "DB80_Label".E1 := "On" AND ("DB80_Label".E1 OR "DB22_DisplayData".dbx23_3);
   "DB80_Label".E2 := "On" AND ("DB80_Label".E2 OR "DB22_DisplayData".dbx23_4);
   "DB80_Label".E3 := "On" AND ("DB80_Label".E3 OR "DB22_DisplayData".dbx23_5);
END_REGION

REGION Network 2: First label apply
   RUNG wire#powerrail
      Contact( "DB80_Label".Step0 )
      Contact( "Auto" )
      wire#w1
      Contact( "DB09_TablePos".Req1_Pos )
      I_Contact( "Timer".T10.Q )
      wire#w2
      S_Coil( "DB80_Label".Step1 )
   END_RUNG
   RUNG wire#w1
      I_Contact( "DB80_Label".Phase1_On )
   END_RUNG wire#w2
   RUNG wire#w2
      R_Coil( "DB80_Label".Step0 )
   END_RUNG
   // the same network as SCL:
   IF "DB80_Label".Step0 AND "Auto" AND (("DB09_TablePos".Req1_Pos AND NOT "Timer".T10.Q) OR NOT "DB80_Label".Phase1_On) THEN
       "DB80_Label".Step1 := TRUE;
       "DB80_Label".Step0 := FALSE;
   END_IF;
END_REGION

REGION Network 3: Table rotation to second label position
   RUNG wire#powerrail
      Contact( "DB80_Label".Step1 )
      Contact( "Auto" )
      wire#w1
      Contact( "DB80_Label".E1 )
      Contact( "DB80_Label".E2 )
      I_Contact( "DB09_TablePos".Req1_Pos )
      wire#w2
      S_Coil( "DB80_Label".Step2 )
   END_RUNG
   RUNG wire#w1
      I_Contact( "DB80_Label".Phase1_On )
   END_RUNG wire#w2
   RUNG wire#w2
      R_Coil( "DB80_Label".Step1 )
   END_RUNG
   // the same network as SCL:
   IF "DB80_Label".Step1 AND "Auto" AND (("DB80_Label".E1 AND "DB80_Label".E2 AND NOT "DB09_TablePos".Req1_Pos) OR NOT "DB80_Label".Phase1_On) THEN
       "DB80_Label".Step2 := TRUE;
       "DB80_Label".Step1 := FALSE;
   END_IF;
END_REGION

REGION Network 4: Second label apply
   RUNG wire#powerrail
      Contact( "DB80_Label".Step2 )
      Contact( "Auto" )
      wire#w1
      Contact( "DB09_TablePos".Req1_Pos )
      I_Contact( "Timer".T10.Q )
      wire#w2
      S_Coil( "DB80_Label".Step3 )
   END_RUNG
   RUNG wire#w1
      I_Contact( "DB80_Label".Phase2_On )
   END_RUNG wire#w2
   RUNG wire#w2
      R_Coil( "DB80_Label".Step2 )
   END_RUNG
   // the same network as SCL:
   IF "DB80_Label".Step2 AND "Auto" AND (("DB09_TablePos".Req1_Pos AND NOT "Timer".T10.Q) OR NOT "DB80_Label".Phase2_On) THEN
       "DB80_Label".Step3 := TRUE;
       "DB80_Label".Step2 := FALSE;
   END_IF;
END_REGION

REGION Network 5: Table rotation to third label position
   RUNG wire#powerrail
      Contact( "DB80_Label".Step3 )
      Contact( "Auto" )
      wire#w1
      Contact( "DB80_Label".E1 )
      Contact( "DB80_Label".E2 )
      I_Contact( "DB09_TablePos".Req1_Pos )
      wire#w2
      S_Coil( "DB80_Label".Step4 )
   END_RUNG
   RUNG wire#w1
      I_Contact( "DB80_Label".Phase2_On )
   END_RUNG wire#w2
   RUNG wire#w2
      R_Coil( "DB80_Label".Step3 )
   END_RUNG
   // the same network as SCL:
   IF "DB80_Label".Step3 AND "Auto" AND (("DB80_Label".E1 AND "DB80_Label".E2 AND NOT "DB09_TablePos".Req1_Pos) OR NOT "DB80_Label".Phase2_On) THEN
       "DB80_Label".Step4 := TRUE;
       "DB80_Label".Step3 := FALSE;
   END_IF;
END_REGION

REGION Network 6: Second label apply
   RUNG wire#powerrail
      Contact( "DB80_Label".Step4 )
      Contact( "Auto" )
      wire#w1
      Contact( "DB09_TablePos".Req1_Pos )
      I_Contact( "Timer".T10.Q )
      wire#w2
      S_Coil( "DB80_Label".Step5 )
   END_RUNG
   RUNG wire#w1
      I_Contact( "DB80_Label".Phase3_On )
   END_RUNG wire#w2
   RUNG wire#w2
      R_Coil( "DB80_Label".Step4 )
   END_RUNG
   // the same network as SCL:
   IF "DB80_Label".Step4 AND "Auto" AND (("DB09_TablePos".Req1_Pos AND NOT "Timer".T10.Q) OR NOT "DB80_Label".Phase3_On) THEN
       "DB80_Label".Step5 := TRUE;
       "DB80_Label".Step4 := FALSE;
   END_IF;
END_REGION

REGION Network 7: Table rotation to fourth label position
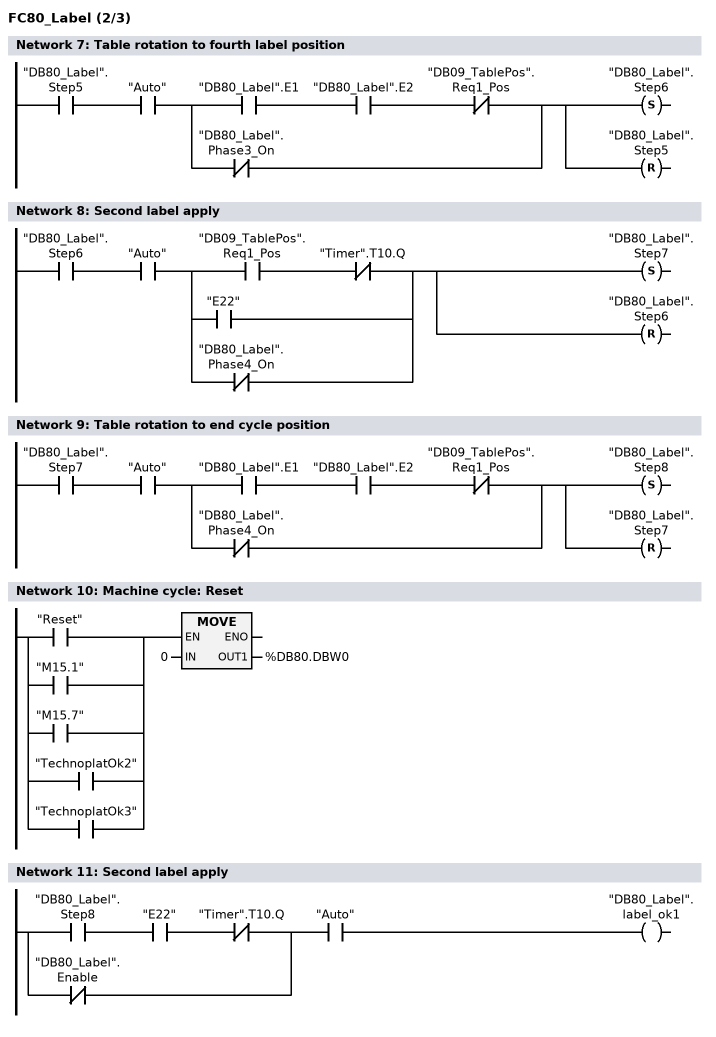
   RUNG wire#powerrail
      Contact( "DB80_Label".Step5 )
      Contact( "Auto" )
      wire#w1
      Contact( "DB80_Label".E1 )
      Contact( "DB80_Label".E2 )
      I_Contact( "DB09_TablePos".Req1_Pos )
      wire#w2
      S_Coil( "DB80_Label".Step6 )
   END_RUNG
   RUNG wire#w1
      I_Contact( "DB80_Label".Phase3_On )
   END_RUNG wire#w2
   RUNG wire#w2
      R_Coil( "DB80_Label".Step5 )
   END_RUNG
   // the same network as SCL:
   IF "DB80_Label".Step5 AND "Auto" AND (("DB80_Label".E1 AND "DB80_Label".E2 AND NOT "DB09_TablePos".Req1_Pos) OR NOT "DB80_Label".Phase3_On) THEN
       "DB80_Label".Step6 := TRUE;
       "DB80_Label".Step5 := FALSE;
   END_IF;
END_REGION

REGION Network 8: Second label apply
   RUNG wire#powerrail
      Contact( "DB80_Label".Step6 )
      Contact( "Auto" )
      wire#w1
      Contact( "DB09_TablePos".Req1_Pos )
      I_Contact( "Timer".T10.Q )
      wire#w2
      S_Coil( "DB80_Label".Step7 )
   END_RUNG
   RUNG wire#w1
      Contact( "E22" )
   END_RUNG wire#w2
   RUNG wire#w1
      I_Contact( "DB80_Label".Phase4_On )
   END_RUNG wire#w2
   RUNG wire#w2
      R_Coil( "DB80_Label".Step6 )
   END_RUNG
   // the same network as SCL:
   IF "DB80_Label".Step6 AND "Auto" AND (("DB09_TablePos".Req1_Pos AND NOT "Timer".T10.Q) OR "E22" OR NOT "DB80_Label".Phase4_On) THEN
       "DB80_Label".Step7 := TRUE;
       "DB80_Label".Step6 := FALSE;
   END_IF;
END_REGION

REGION Network 9: Table rotation to end cycle position
   RUNG wire#powerrail
      Contact( "DB80_Label".Step7 )
      Contact( "Auto" )
      wire#w1
      Contact( "DB80_Label".E1 )
      Contact( "DB80_Label".E2 )
      I_Contact( "DB09_TablePos".Req1_Pos )
      wire#w2
      S_Coil( "DB80_Label".Step8 )
   END_RUNG
   RUNG wire#w1
      I_Contact( "DB80_Label".Phase4_On )
   END_RUNG wire#w2
   RUNG wire#w2
      R_Coil( "DB80_Label".Step7 )
   END_RUNG
   // the same network as SCL:
   IF "DB80_Label".Step7 AND "Auto" AND (("DB80_Label".E1 AND "DB80_Label".E2 AND NOT "DB09_TablePos".Req1_Pos) OR NOT "DB80_Label".Phase4_On) THEN
       "DB80_Label".Step8 := TRUE;
       "DB80_Label".Step7 := FALSE;
   END_IF;
END_REGION

REGION Network 10: Machine cycle: Reset
   RUNG wire#powerrail
      Contact( "Reset" )
      wire#w1
      { S7_GenerateENO := "TRUE" } Move(in := 0, out1 => %DB80.DBW0)
   END_RUNG
   RUNG wire#powerrail
      Contact( "M15.1" )
   END_RUNG wire#w1
   RUNG wire#powerrail
      Contact( "M15.7" )
   END_RUNG wire#w1
   RUNG wire#powerrail
      Contact( "TechnoplatOk2" )
   END_RUNG wire#w1
   RUNG wire#powerrail
      Contact( "TechnoplatOk3" )
   END_RUNG wire#w1
   // the same network as SCL:
   IF "Reset" OR "M15.1" OR "M15.7" OR "TechnoplatOk2" OR "TechnoplatOk3" THEN %DB80.DBW0 := 0; END_IF;
END_REGION

REGION Network 11: Second label apply
   RUNG wire#powerrail
      Contact( "DB80_Label".Step8 )
      Contact( "E22" )
      I_Contact( "Timer".T10.Q )
      wire#w1
      Contact( "Auto" )
      Coil( "DB80_Label".label_ok1 )
   END_RUNG
   RUNG wire#powerrail
      I_Contact( "DB80_Label".Enable )
   END_RUNG wire#w1
   // the same network as SCL:
   "DB80_Label".label_ok1 := (("DB80_Label".Step8 AND "E22" AND NOT "Timer".T10.Q) OR NOT "DB80_Label".Enable) AND "Auto";
END_REGION

REGION Network 12: Label phases
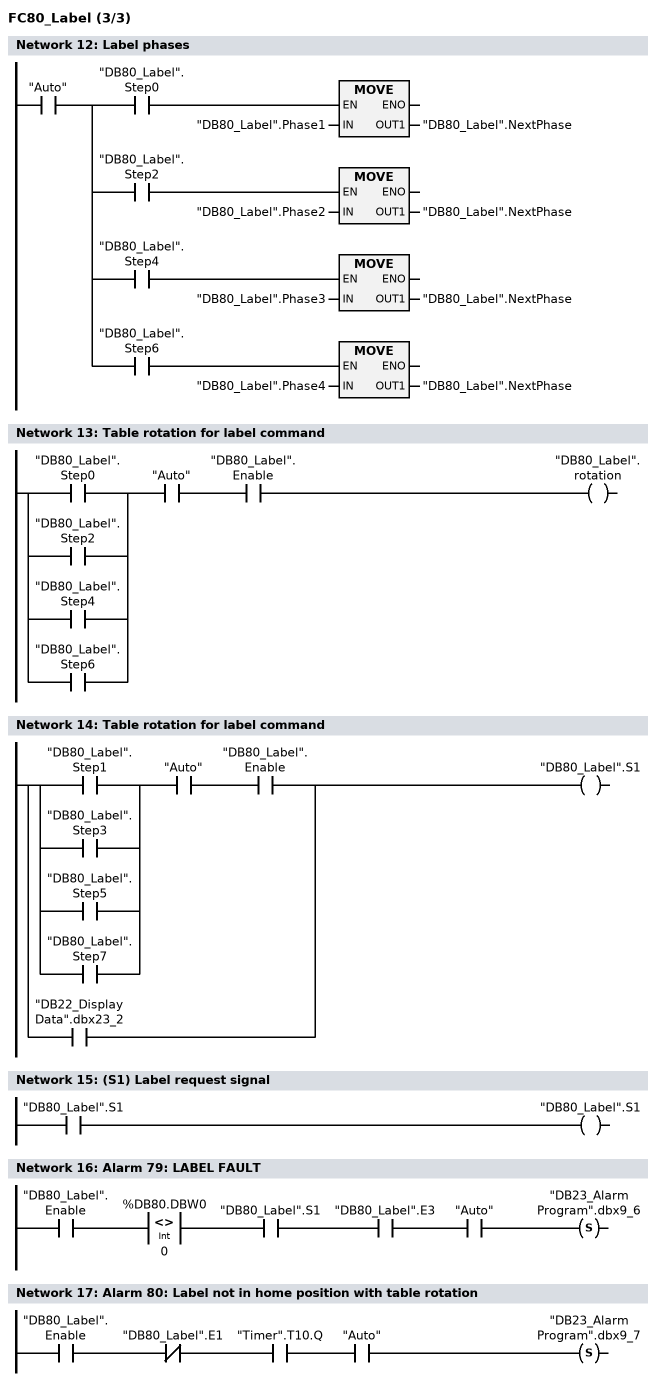
   RUNG wire#powerrail
      Contact( "Auto" )
      wire#w1
      Contact( "DB80_Label".Step0 )
      { S7_GenerateENO := "TRUE" } Move(in := "DB80_Label".Phase1, out1 => "DB80_Label".NextPhase)
   END_RUNG
   RUNG wire#w1
      Contact( "DB80_Label".Step2 )
      { S7_GenerateENO := "TRUE" } Move(in := "DB80_Label".Phase2, out1 => "DB80_Label".NextPhase)
   END_RUNG
   RUNG wire#w1
      Contact( "DB80_Label".Step4 )
      { S7_GenerateENO := "TRUE" } Move(in := "DB80_Label".Phase3, out1 => "DB80_Label".NextPhase)
   END_RUNG
   RUNG wire#w1
      Contact( "DB80_Label".Step6 )
      { S7_GenerateENO := "TRUE" } Move(in := "DB80_Label".Phase4, out1 => "DB80_Label".NextPhase)
   END_RUNG
   // the same network as SCL:
   IF "Auto" AND "DB80_Label".Step0 THEN "DB80_Label".NextPhase := "DB80_Label".Phase1; END_IF;
   IF "Auto" AND "DB80_Label".Step2 THEN "DB80_Label".NextPhase := "DB80_Label".Phase2; END_IF;
   IF "Auto" AND "DB80_Label".Step4 THEN "DB80_Label".NextPhase := "DB80_Label".Phase3; END_IF;
   IF "Auto" AND "DB80_Label".Step6 THEN "DB80_Label".NextPhase := "DB80_Label".Phase4; END_IF;
END_REGION

REGION Network 13: Table rotation for label command
   RUNG wire#powerrail
      Contact( "DB80_Label".Step0 )
      wire#w1
      Contact( "Auto" )
      Contact( "DB80_Label".Enable )
      Coil( "DB80_Label".rotation )
   END_RUNG
   RUNG wire#powerrail
      Contact( "DB80_Label".Step2 )
   END_RUNG wire#w1
   RUNG wire#powerrail
      Contact( "DB80_Label".Step4 )
   END_RUNG wire#w1
   RUNG wire#powerrail
      Contact( "DB80_Label".Step6 )
   END_RUNG wire#w1
   // the same network as SCL:
   "DB80_Label".rotation := ("DB80_Label".Step0 OR "DB80_Label".Step2 OR "DB80_Label".Step4 OR "DB80_Label".Step6) AND "Auto" AND "DB80_Label".Enable;
END_REGION

REGION Network 14: Table rotation for label command
   RUNG wire#powerrail
      Contact( "DB80_Label".Step1 )
      wire#w1
      Contact( "Auto" )
      Contact( "DB80_Label".Enable )
      wire#w2
      Coil( "DB80_Label".S1 )
   END_RUNG
   RUNG wire#powerrail
      Contact( "DB80_Label".Step3 )
   END_RUNG wire#w1
   RUNG wire#powerrail
      Contact( "DB80_Label".Step5 )
   END_RUNG wire#w1
   RUNG wire#powerrail
      Contact( "DB80_Label".Step7 )
   END_RUNG wire#w1
   RUNG wire#powerrail
      Contact( "DB22_DisplayData".dbx23_2 )
   END_RUNG wire#w2
   // the same network as SCL:
   "DB80_Label".S1 := (("DB80_Label".Step1 OR "DB80_Label".Step3 OR "DB80_Label".Step5 OR "DB80_Label".Step7) AND "Auto" AND "DB80_Label".Enable) OR "DB22_DisplayData".dbx23_2;
END_REGION

REGION Network 15: (S1) Label request signal
   RUNG wire#powerrail
      Contact( "DB80_Label".S1 )
      Coil( "DB80_Label".S1 )
   END_RUNG
   // the same network as SCL:
   "DB80_Label".S1 := "DB80_Label".S1;
END_REGION

REGION Network 16: Alarm 79: LABEL FAULT
   RUNG wire#powerrail
      Contact( "DB80_Label".Enable )
      { S7_Templates := "SrcType := Int" } NE_Contact(in1 := %DB80.DBW0, in2 := 0)
      Contact( "DB80_Label".S1 )
      Contact( "DB80_Label".E3 )
      Contact( "Auto" )
      S_Coil( "DB23_AlarmProgram".dbx9_6 )
   END_RUNG
   // the same network as SCL:
   IF "DB80_Label".Enable AND (%DB80.DBW0 <> 0) AND "DB80_Label".S1 AND "DB80_Label".E3 AND "Auto" THEN
       "DB23_AlarmProgram".dbx9_6 := TRUE;
   END_IF;
END_REGION

REGION Network 17: Alarm 80: Label not in home position with table rotation
   RUNG wire#powerrail
      Contact( "DB80_Label".Enable )
      I_Contact( "DB80_Label".E1 )
      Contact( "Timer".T10.Q )
      Contact( "Auto" )
      S_Coil( "DB23_AlarmProgram".dbx9_7 )
   END_RUNG
   // the same network as SCL:
   IF "DB80_Label".Enable AND NOT "DB80_Label".E1 AND "Timer".T10.Q AND "Auto" THEN
       "DB23_AlarmProgram".dbx9_7 := TRUE;
   END_IF;
END_REGION
END_FUNCTION

FUNCTION "FC86_Conveyor_5_IN_3_OUT" : Void   // FC86, LAD
TITLE = Conveyor_5_IN_3_OUT
{ S7_Optimized_Access := 'TRUE' }
VERSION : 0.1
// 5+3 (Fitembal)
// stored: AutoNumber false, IsIECCheckEnabled false, SetENOAutomatically false, UDAEnableTagReadback false
   VAR_TEMP   // added for the SCL form of the ladder/FBD networks
      _w1 : Bool;
      _w2 : Bool;
   END_VAR
BEGIN

REGION Network 1: Manual operation for conveyor
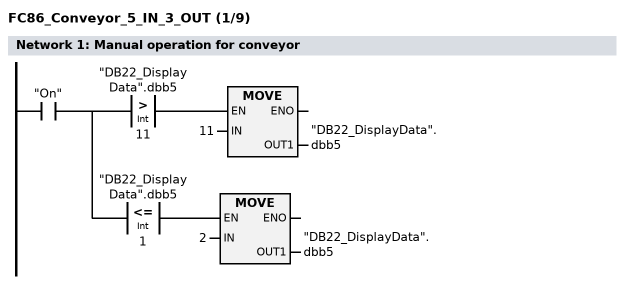
   RUNG wire#powerrail
      Contact( "On" )
      wire#w1
      { S7_Templates := "SrcType := Int" } GT_Contact(in1 := "DB22_DisplayData".dbb5, in2 := 11)
      { S7_GenerateENO := "TRUE" } Move(in := 11, out1 => "DB22_DisplayData".dbb5)
   END_RUNG
   RUNG wire#w1
      { S7_Templates := "SrcType := Int" } LE_Contact(in1 := "DB22_DisplayData".dbb5, in2 := 1)
      { S7_GenerateENO := "TRUE" } Move(in := 2, out1 => "DB22_DisplayData".dbb5)
   END_RUNG
   // the same network as SCL:
   IF "On" AND ("DB22_DisplayData".dbb5 > 11) THEN "DB22_DisplayData".dbb5 := 11; END_IF;
   IF "On" AND ("DB22_DisplayData".dbb5 <= 1) THEN "DB22_DisplayData".dbb5 := 2; END_IF;
END_REGION

REGION Network 2: Manual operation for conveyor
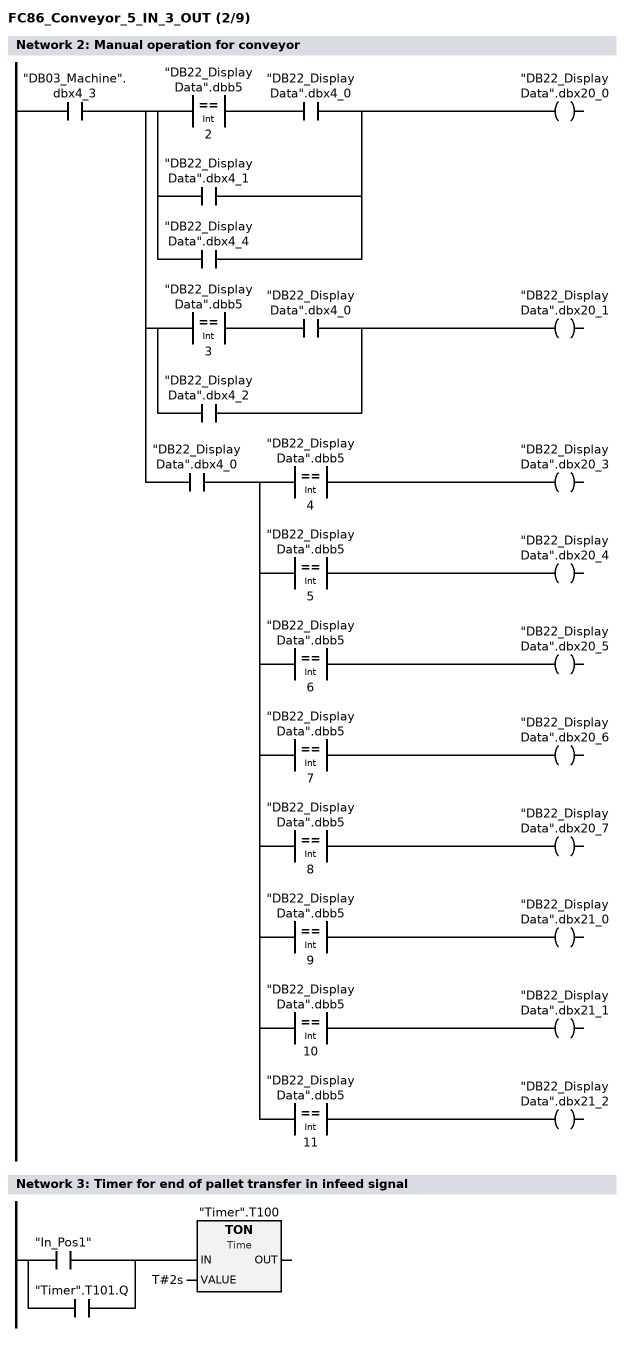
   RUNG wire#powerrail
      Contact( "DB03_Machine".dbx4_3 )
      wire#w1
      { S7_Templates := "SrcType := Int" } EQ_Contact(in1 := "DB22_DisplayData".dbb5, in2 := 2)
      Contact( "DB22_DisplayData".dbx4_0 )
      wire#w2
      Coil( "DB22_DisplayData".dbx20_0 )
   END_RUNG
   RUNG wire#w1
      Contact( "DB22_DisplayData".dbx4_1 )
   END_RUNG wire#w2
   RUNG wire#w1
      Contact( "DB22_DisplayData".dbx4_4 )
   END_RUNG wire#w2
   RUNG wire#w1
      { S7_Templates := "SrcType := Int" } EQ_Contact(in1 := "DB22_DisplayData".dbb5, in2 := 3)
      Contact( "DB22_DisplayData".dbx4_0 )
      wire#w3
      Coil( "DB22_DisplayData".dbx20_1 )
   END_RUNG
   RUNG wire#w1
      Contact( "DB22_DisplayData".dbx4_2 )
   END_RUNG wire#w3
   RUNG wire#w1
      Contact( "DB22_DisplayData".dbx4_0 )
      wire#w4
      { S7_Templates := "SrcType := Int" } EQ_Contact(in1 := "DB22_DisplayData".dbb5, in2 := 4)
      Coil( "DB22_DisplayData".dbx20_3 )
   END_RUNG
   RUNG wire#w4
      { S7_Templates := "SrcType := Int" } EQ_Contact(in1 := "DB22_DisplayData".dbb5, in2 := 5)
      Coil( "DB22_DisplayData".dbx20_4 )
   END_RUNG
   RUNG wire#w4
      { S7_Templates := "SrcType := Int" } EQ_Contact(in1 := "DB22_DisplayData".dbb5, in2 := 6)
      Coil( "DB22_DisplayData".dbx20_5 )
   END_RUNG
   RUNG wire#w4
      { S7_Templates := "SrcType := Int" } EQ_Contact(in1 := "DB22_DisplayData".dbb5, in2 := 7)
      Coil( "DB22_DisplayData".dbx20_6 )
   END_RUNG
   RUNG wire#w4
      { S7_Templates := "SrcType := Int" } EQ_Contact(in1 := "DB22_DisplayData".dbb5, in2 := 8)
      Coil( "DB22_DisplayData".dbx20_7 )
   END_RUNG
   RUNG wire#w4
      { S7_Templates := "SrcType := Int" } EQ_Contact(in1 := "DB22_DisplayData".dbb5, in2 := 9)
      Coil( "DB22_DisplayData".dbx21_0 )
   END_RUNG
   RUNG wire#w4
      { S7_Templates := "SrcType := Int" } EQ_Contact(in1 := "DB22_DisplayData".dbb5, in2 := 10)
      Coil( "DB22_DisplayData".dbx21_1 )
   END_RUNG
   RUNG wire#w4
      { S7_Templates := "SrcType := Int" } EQ_Contact(in1 := "DB22_DisplayData".dbb5, in2 := 11)
      Coil( "DB22_DisplayData".dbx21_2 )
   END_RUNG
   // the same network as SCL:
   "DB22_DisplayData".dbx20_0 := "DB03_Machine".dbx4_3 AND ((("DB22_DisplayData".dbb5 = 2) AND "DB22_DisplayData".dbx4_0) OR "DB22_DisplayData".dbx4_1 OR "DB22_DisplayData".dbx4_4);
   "DB22_DisplayData".dbx20_1 := "DB03_Machine".dbx4_3 AND ((("DB22_DisplayData".dbb5 = 3) AND "DB22_DisplayData".dbx4_0) OR "DB22_DisplayData".dbx4_2);
   #_w1 := "DB03_Machine".dbx4_3 AND "DB22_DisplayData".dbx4_0;
   "DB22_DisplayData".dbx20_3 := #_w1 AND ("DB22_DisplayData".dbb5 = 4);
   "DB22_DisplayData".dbx20_4 := #_w1 AND ("DB22_DisplayData".dbb5 = 5);
   "DB22_DisplayData".dbx20_5 := #_w1 AND ("DB22_DisplayData".dbb5 = 6);
   "DB22_DisplayData".dbx20_6 := #_w1 AND ("DB22_DisplayData".dbb5 = 7);
   "DB22_DisplayData".dbx20_7 := #_w1 AND ("DB22_DisplayData".dbb5 = 8);
   "DB22_DisplayData".dbx21_0 := #_w1 AND ("DB22_DisplayData".dbb5 = 9);
   "DB22_DisplayData".dbx21_1 := #_w1 AND ("DB22_DisplayData".dbb5 = 10);
   "DB22_DisplayData".dbx21_2 := #_w1 AND ("DB22_DisplayData".dbb5 = 11);
END_REGION

REGION Network 3: Timer for end of pallet transfer in infeed signal
   "Timer".T100.TON(IN := "In_Pos1" OR "Timer".T101.Q, PT := T#2s);   // TON coil
END_REGION

REGION Network 4: Timeout for conveyor pos1
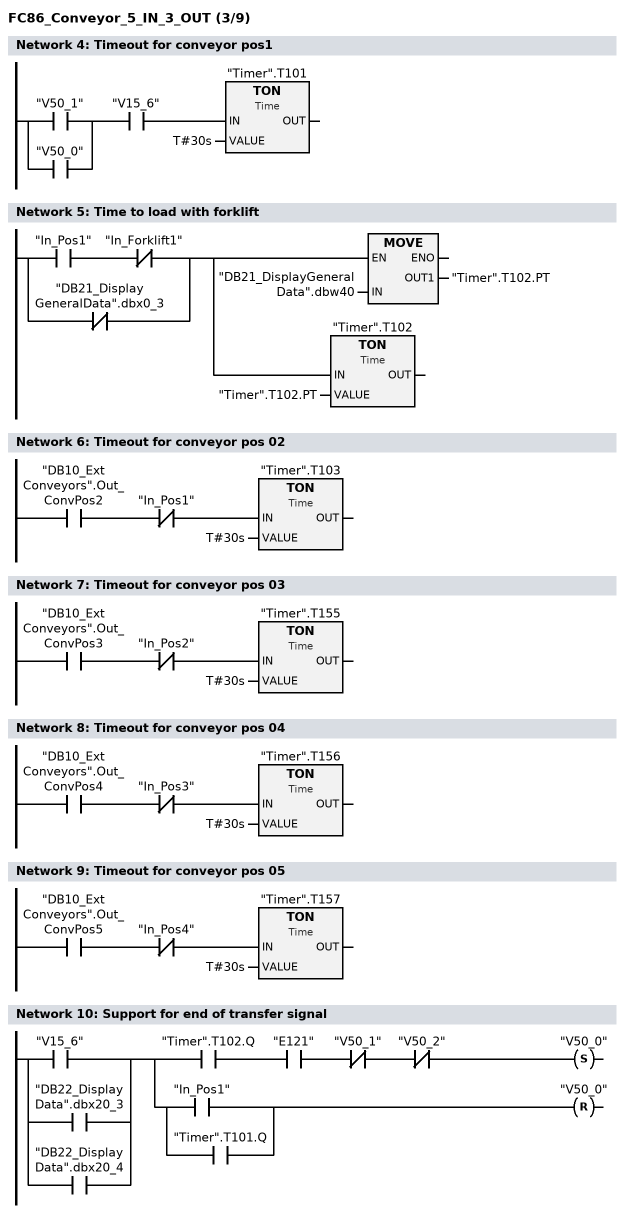
   "Timer".T101.TON(IN := ("V50_1" OR "V50_0") AND "V15_6", PT := T#30s);   // TON coil
END_REGION

REGION Network 5: Time to load with forklift
   #_w1 := ("In_Pos1" AND NOT "In_Forklift1") OR NOT "DB21_DisplayGeneralData".dbx0_3;
   IF #_w1 THEN "Timer".T102.PT := "DB21_DisplayGeneralData".dbw40; END_IF;
   "Timer".T102.TON(IN := #_w1, PT := "Timer".T102.PT);   // TON coil
END_REGION

REGION Network 6: Timeout for conveyor pos 02
   "Timer".T103.TON(IN := "DB10_ExtConveyors".Out_ConvPos2 AND NOT "In_Pos1", PT := T#30s);   // TON coil
END_REGION

REGION Network 7: Timeout for conveyor pos 03
   "Timer".T155.TON(IN := "DB10_ExtConveyors".Out_ConvPos3 AND NOT "In_Pos2", PT := T#30s);   // TON coil
END_REGION

REGION Network 8: Timeout for conveyor pos 04
   "Timer".T156.TON(IN := "DB10_ExtConveyors".Out_ConvPos4 AND NOT "In_Pos3", PT := T#30s);   // TON coil
END_REGION

REGION Network 9: Timeout for conveyor pos 05
   "Timer".T157.TON(IN := "DB10_ExtConveyors".Out_ConvPos5 AND NOT "In_Pos4", PT := T#30s);   // TON coil
END_REGION

REGION Network 10: Support for end of transfer signal
   RUNG wire#powerrail
      Contact( "V15_6" )
      wire#w1
      Contact( "Timer".T102.Q )
      Contact( "E121" )
      I_Contact( "V50_1" )
      I_Contact( "V50_2" )
      S_Coil( "V50_0" )
   END_RUNG
   RUNG wire#powerrail
      Contact( "DB22_DisplayData".dbx20_3 )
   END_RUNG wire#w1
   RUNG wire#powerrail
      Contact( "DB22_DisplayData".dbx20_4 )
   END_RUNG wire#w1
   RUNG wire#w1
      Contact( "In_Pos1" )
      wire#w2
      R_Coil( "V50_0" )
   END_RUNG
   RUNG wire#w1
      Contact( "Timer".T101.Q )
   END_RUNG wire#w2
   // the same network as SCL:
   #_w1 := "V15_6" OR "DB22_DisplayData".dbx20_3 OR "DB22_DisplayData".dbx20_4;
   IF #_w1 AND "Timer".T102.Q AND "E121" AND NOT "V50_1" AND NOT "V50_2" THEN "V50_0" := TRUE; END_IF;
   IF #_w1 AND ("In_Pos1" OR "Timer".T101.Q) THEN "V50_0" := FALSE; END_IF;
END_REGION

REGION Network 11: Transit memory for conveyor pos1
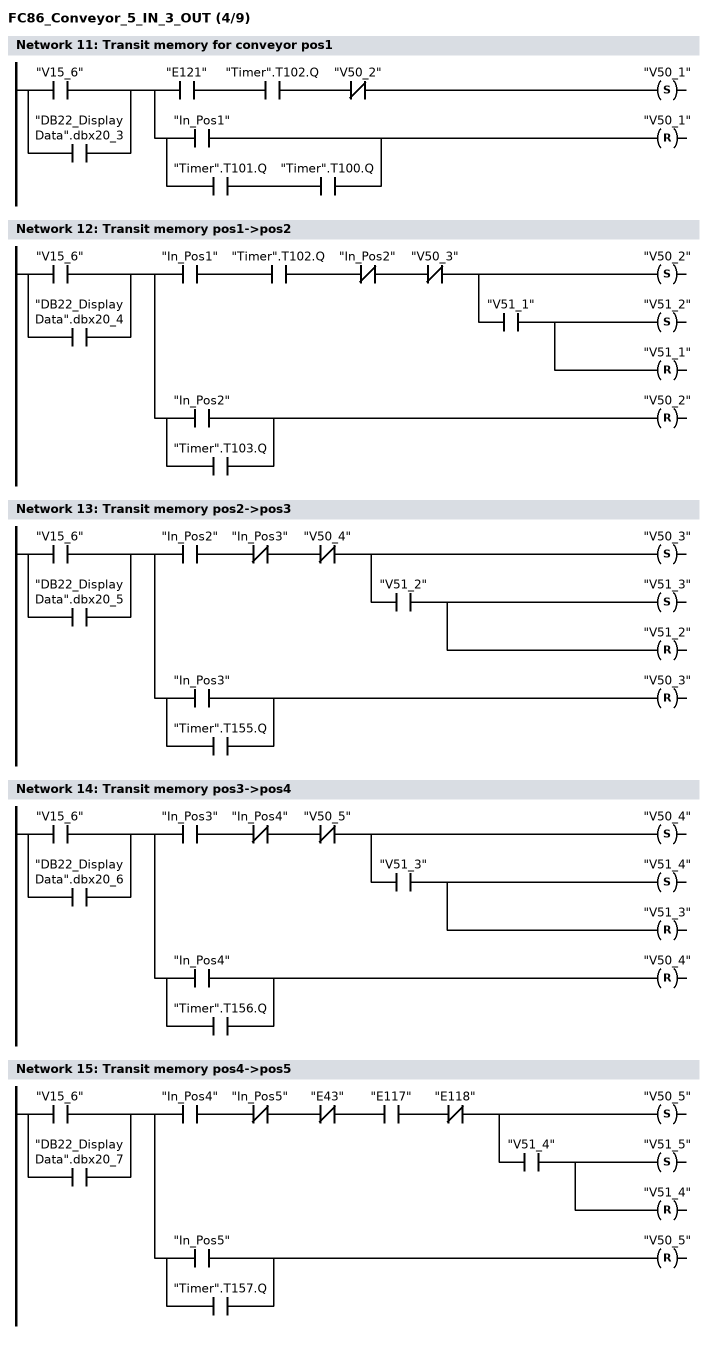
   RUNG wire#powerrail
      Contact( "V15_6" )
      wire#w1
      Contact( "E121" )
      Contact( "Timer".T102.Q )
      I_Contact( "V50_2" )
      S_Coil( "V50_1" )
   END_RUNG
   RUNG wire#powerrail
      Contact( "DB22_DisplayData".dbx20_3 )
   END_RUNG wire#w1
   RUNG wire#w1
      Contact( "In_Pos1" )
      wire#w2
      R_Coil( "V50_1" )
   END_RUNG
   RUNG wire#w1
      Contact( "Timer".T101.Q )
      Contact( "Timer".T100.Q )
   END_RUNG wire#w2
   // the same network as SCL:
   #_w1 := "V15_6" OR "DB22_DisplayData".dbx20_3;
   IF #_w1 AND "E121" AND "Timer".T102.Q AND NOT "V50_2" THEN "V50_1" := TRUE; END_IF;
   IF #_w1 AND ("In_Pos1" OR ("Timer".T101.Q AND "Timer".T100.Q)) THEN "V50_1" := FALSE; END_IF;
END_REGION

REGION Network 12: Transit memory pos1->pos2
   RUNG wire#powerrail
      Contact( "V15_6" )
      wire#w1
      Contact( "In_Pos1" )
      Contact( "Timer".T102.Q )
      I_Contact( "In_Pos2" )
      I_Contact( "V50_3" )
      wire#w2
      S_Coil( "V50_2" )
   END_RUNG
   RUNG wire#powerrail
      Contact( "DB22_DisplayData".dbx20_4 )
   END_RUNG wire#w1
   RUNG wire#w2
      Contact( "V51_1" )
      wire#w3
      S_Coil( "V51_2" )
   END_RUNG
   RUNG wire#w3
      R_Coil( "V51_1" )
   END_RUNG
   RUNG wire#w1
      Contact( "In_Pos2" )
      wire#w4
      R_Coil( "V50_2" )
   END_RUNG
   RUNG wire#w1
      Contact( "Timer".T103.Q )
   END_RUNG wire#w4
   // the same network as SCL:
   #_w1 := "V15_6" OR "DB22_DisplayData".dbx20_4;
   #_w2 := #_w1 AND "In_Pos1" AND "Timer".T102.Q AND NOT "In_Pos2" AND NOT "V50_3";
   IF #_w2 THEN "V50_2" := TRUE; END_IF;
   IF #_w2 AND "V51_1" THEN
       "V51_2" := TRUE;
       "V51_1" := FALSE;
   END_IF;
   IF #_w1 AND ("In_Pos2" OR "Timer".T103.Q) THEN "V50_2" := FALSE; END_IF;
END_REGION

REGION Network 13: Transit memory pos2->pos3
   RUNG wire#powerrail
      Contact( "V15_6" )
      wire#w1
      Contact( "In_Pos2" )
      I_Contact( "In_Pos3" )
      I_Contact( "V50_4" )
      wire#w2
      S_Coil( "V50_3" )
   END_RUNG
   RUNG wire#powerrail
      Contact( "DB22_DisplayData".dbx20_5 )
   END_RUNG wire#w1
   RUNG wire#w2
      Contact( "V51_2" )
      wire#w3
      S_Coil( "V51_3" )
   END_RUNG
   RUNG wire#w3
      R_Coil( "V51_2" )
   END_RUNG
   RUNG wire#w1
      Contact( "In_Pos3" )
      wire#w4
      R_Coil( "V50_3" )
   END_RUNG
   RUNG wire#w1
      Contact( "Timer".T155.Q )
   END_RUNG wire#w4
   // the same network as SCL:
   #_w1 := "V15_6" OR "DB22_DisplayData".dbx20_5;
   #_w2 := #_w1 AND "In_Pos2" AND NOT "In_Pos3" AND NOT "V50_4";
   IF #_w2 THEN "V50_3" := TRUE; END_IF;
   IF #_w2 AND "V51_2" THEN
       "V51_3" := TRUE;
       "V51_2" := FALSE;
   END_IF;
   IF #_w1 AND ("In_Pos3" OR "Timer".T155.Q) THEN "V50_3" := FALSE; END_IF;
END_REGION

REGION Network 14: Transit memory pos3->pos4
   RUNG wire#powerrail
      Contact( "V15_6" )
      wire#w1
      Contact( "In_Pos3" )
      I_Contact( "In_Pos4" )
      I_Contact( "V50_5" )
      wire#w2
      S_Coil( "V50_4" )
   END_RUNG
   RUNG wire#powerrail
      Contact( "DB22_DisplayData".dbx20_6 )
   END_RUNG wire#w1
   RUNG wire#w2
      Contact( "V51_3" )
      wire#w3
      S_Coil( "V51_4" )
   END_RUNG
   RUNG wire#w3
      R_Coil( "V51_3" )
   END_RUNG
   RUNG wire#w1
      Contact( "In_Pos4" )
      wire#w4
      R_Coil( "V50_4" )
   END_RUNG
   RUNG wire#w1
      Contact( "Timer".T156.Q )
   END_RUNG wire#w4
   // the same network as SCL:
   #_w1 := "V15_6" OR "DB22_DisplayData".dbx20_6;
   #_w2 := #_w1 AND "In_Pos3" AND NOT "In_Pos4" AND NOT "V50_5";
   IF #_w2 THEN "V50_4" := TRUE; END_IF;
   IF #_w2 AND "V51_3" THEN
       "V51_4" := TRUE;
       "V51_3" := FALSE;
   END_IF;
   IF #_w1 AND ("In_Pos4" OR "Timer".T156.Q) THEN "V50_4" := FALSE; END_IF;
END_REGION

REGION Network 15: Transit memory pos4->pos5
   RUNG wire#powerrail
      Contact( "V15_6" )
      wire#w1
      Contact( "In_Pos4" )
      I_Contact( "In_Pos5" )
      I_Contact( "E43" )
      Contact( "E117" )
      I_Contact( "E118" )
      wire#w2
      S_Coil( "V50_5" )
   END_RUNG
   RUNG wire#powerrail
      Contact( "DB22_DisplayData".dbx20_7 )
   END_RUNG wire#w1
   RUNG wire#w2
      Contact( "V51_4" )
      wire#w3
      S_Coil( "V51_5" )
   END_RUNG
   RUNG wire#w3
      R_Coil( "V51_4" )
   END_RUNG
   RUNG wire#w1
      Contact( "In_Pos5" )
      wire#w4
      R_Coil( "V50_5" )
   END_RUNG
   RUNG wire#w1
      Contact( "Timer".T157.Q )
   END_RUNG wire#w4
   // the same network as SCL:
   #_w1 := "V15_6" OR "DB22_DisplayData".dbx20_7;
   #_w2 := #_w1 AND "In_Pos4" AND NOT "In_Pos5" AND NOT "E43" AND "E117" AND NOT "E118";
   IF #_w2 THEN "V50_5" := TRUE; END_IF;
   IF #_w2 AND "V51_4" THEN
       "V51_5" := TRUE;
       "V51_4" := FALSE;
   END_IF;
   IF #_w1 AND ("In_Pos5" OR "Timer".T157.Q) THEN "V50_5" := FALSE; END_IF;
END_REGION

REGION Network 16: Ready to receive pallet in infeed signal
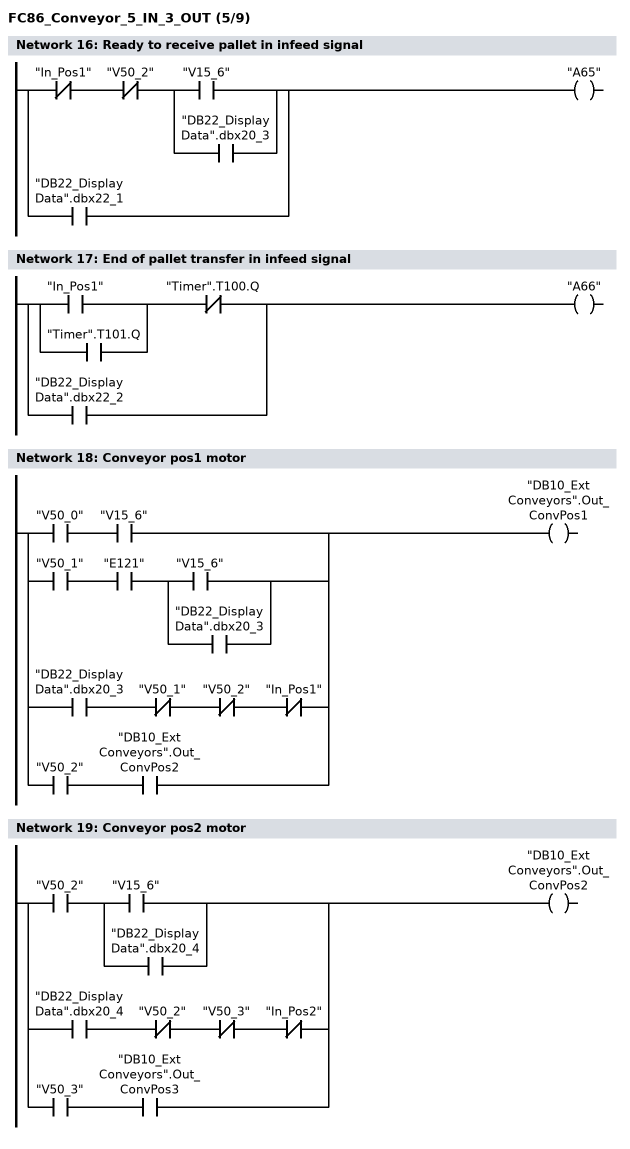
   RUNG wire#powerrail
      I_Contact( "In_Pos1" )
      I_Contact( "V50_2" )
      wire#w1
      Contact( "V15_6" )
      wire#w2
      Coil( "A65" )
   END_RUNG
   RUNG wire#w1
      Contact( "DB22_DisplayData".dbx20_3 )
   END_RUNG wire#w2
   RUNG wire#powerrail
      Contact( "DB22_DisplayData".dbx22_1 )
   END_RUNG wire#w2
   // the same network as SCL:
   "A65" := (NOT "In_Pos1" AND NOT "V50_2" AND ("V15_6" OR "DB22_DisplayData".dbx20_3)) OR "DB22_DisplayData".dbx22_1;
END_REGION

REGION Network 17: End of pallet transfer in infeed signal
   RUNG wire#powerrail
      Contact( "In_Pos1" )
      wire#w1
      I_Contact( "Timer".T100.Q )
      wire#w2
      Coil( "A66" )
   END_RUNG
   RUNG wire#powerrail
      Contact( "Timer".T101.Q )
   END_RUNG wire#w1
   RUNG wire#powerrail
      Contact( "DB22_DisplayData".dbx22_2 )
   END_RUNG wire#w2
   // the same network as SCL:
   "A66" := (("In_Pos1" OR "Timer".T101.Q) AND NOT "Timer".T100.Q) OR "DB22_DisplayData".dbx22_2;
END_REGION

REGION Network 18: Conveyor pos1 motor
   RUNG wire#powerrail
      Contact( "V50_0" )
      Contact( "V15_6" )
      wire#w1
      Coil( "DB10_ExtConveyors".Out_ConvPos1 )
   END_RUNG
   RUNG wire#powerrail
      Contact( "V50_1" )
      Contact( "E121" )
      wire#w2
      Contact( "V15_6" )
   END_RUNG wire#w1
   RUNG wire#w2
      Contact( "DB22_DisplayData".dbx20_3 )
   END_RUNG wire#w1
   RUNG wire#powerrail
      Contact( "DB22_DisplayData".dbx20_3 )
      I_Contact( "V50_1" )
      I_Contact( "V50_2" )
      I_Contact( "In_Pos1" )
   END_RUNG wire#w1
   RUNG wire#powerrail
      Contact( "V50_2" )
      Contact( "DB10_ExtConveyors".Out_ConvPos2 )
   END_RUNG wire#w1
   // the same network as SCL:
   "DB10_ExtConveyors".Out_ConvPos1 := ("V50_0" AND "V15_6") OR ("V50_1" AND "E121" AND ("V15_6" OR "DB22_DisplayData".dbx20_3)) OR ("DB22_DisplayData".dbx20_3 AND NOT "V50_1" AND NOT "V50_2" AND NOT "In_Pos1") OR ("V50_2" AND "DB10_ExtConveyors".Out_ConvPos2);
END_REGION

REGION Network 19: Conveyor pos2 motor
   RUNG wire#powerrail
      Contact( "V50_2" )
      wire#w1
      Contact( "V15_6" )
      wire#w2
      Coil( "DB10_ExtConveyors".Out_ConvPos2 )
   END_RUNG
   RUNG wire#w1
      Contact( "DB22_DisplayData".dbx20_4 )
   END_RUNG wire#w2
   RUNG wire#powerrail
      Contact( "DB22_DisplayData".dbx20_4 )
      I_Contact( "V50_2" )
      I_Contact( "V50_3" )
      I_Contact( "In_Pos2" )
   END_RUNG wire#w2
   RUNG wire#powerrail
      Contact( "V50_3" )
      Contact( "DB10_ExtConveyors".Out_ConvPos3 )
   END_RUNG wire#w2
   // the same network as SCL:
   "DB10_ExtConveyors".Out_ConvPos2 := ("V50_2" AND ("V15_6" OR "DB22_DisplayData".dbx20_4)) OR ("DB22_DisplayData".dbx20_4 AND NOT "V50_2" AND NOT "V50_3" AND NOT "In_Pos2") OR ("V50_3" AND "DB10_ExtConveyors".Out_ConvPos3);
END_REGION

REGION Network 20: Conveyor pos3 motor
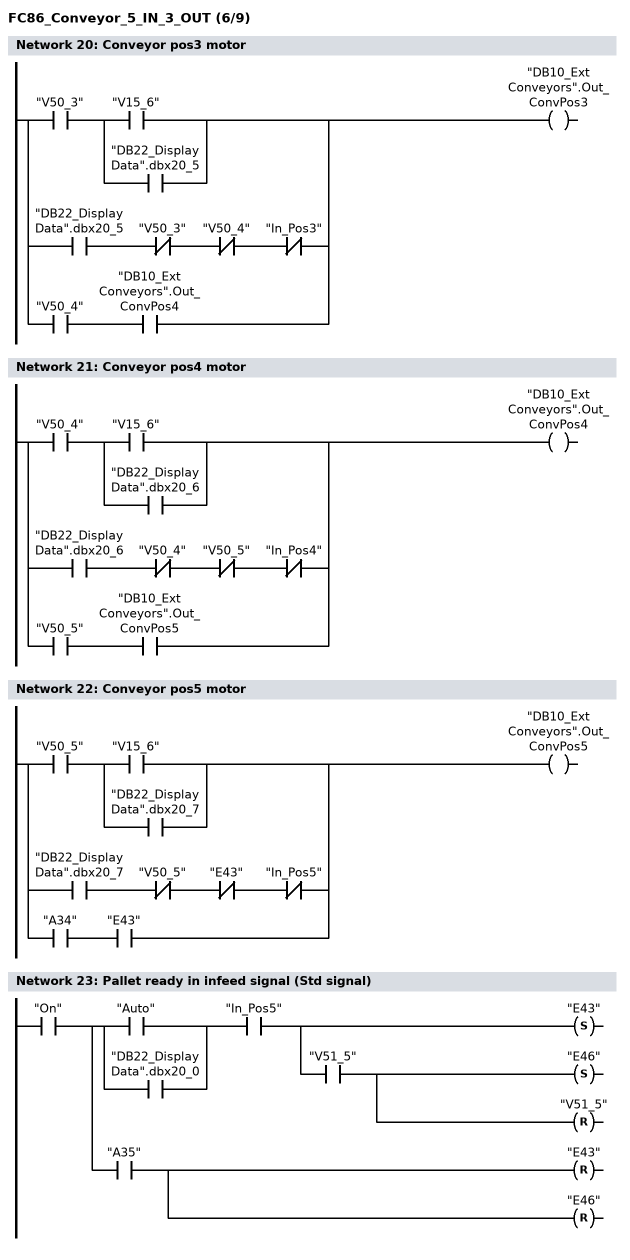
   RUNG wire#powerrail
      Contact( "V50_3" )
      wire#w1
      Contact( "V15_6" )
      wire#w2
      Coil( "DB10_ExtConveyors".Out_ConvPos3 )
   END_RUNG
   RUNG wire#w1
      Contact( "DB22_DisplayData".dbx20_5 )
   END_RUNG wire#w2
   RUNG wire#powerrail
      Contact( "DB22_DisplayData".dbx20_5 )
      I_Contact( "V50_3" )
      I_Contact( "V50_4" )
      I_Contact( "In_Pos3" )
   END_RUNG wire#w2
   RUNG wire#powerrail
      Contact( "V50_4" )
      Contact( "DB10_ExtConveyors".Out_ConvPos4 )
   END_RUNG wire#w2
   // the same network as SCL:
   "DB10_ExtConveyors".Out_ConvPos3 := ("V50_3" AND ("V15_6" OR "DB22_DisplayData".dbx20_5)) OR ("DB22_DisplayData".dbx20_5 AND NOT "V50_3" AND NOT "V50_4" AND NOT "In_Pos3") OR ("V50_4" AND "DB10_ExtConveyors".Out_ConvPos4);
END_REGION

REGION Network 21: Conveyor pos4 motor
   RUNG wire#powerrail
      Contact( "V50_4" )
      wire#w1
      Contact( "V15_6" )
      wire#w2
      Coil( "DB10_ExtConveyors".Out_ConvPos4 )
   END_RUNG
   RUNG wire#w1
      Contact( "DB22_DisplayData".dbx20_6 )
   END_RUNG wire#w2
   RUNG wire#powerrail
      Contact( "DB22_DisplayData".dbx20_6 )
      I_Contact( "V50_4" )
      I_Contact( "V50_5" )
      I_Contact( "In_Pos4" )
   END_RUNG wire#w2
   RUNG wire#powerrail
      Contact( "V50_5" )
      Contact( "DB10_ExtConveyors".Out_ConvPos5 )
   END_RUNG wire#w2
   // the same network as SCL:
   "DB10_ExtConveyors".Out_ConvPos4 := ("V50_4" AND ("V15_6" OR "DB22_DisplayData".dbx20_6)) OR ("DB22_DisplayData".dbx20_6 AND NOT "V50_4" AND NOT "V50_5" AND NOT "In_Pos4") OR ("V50_5" AND "DB10_ExtConveyors".Out_ConvPos5);
END_REGION

REGION Network 22: Conveyor pos5 motor
   RUNG wire#powerrail
      Contact( "V50_5" )
      wire#w1
      Contact( "V15_6" )
      wire#w2
      Coil( "DB10_ExtConveyors".Out_ConvPos5 )
   END_RUNG
   RUNG wire#w1
      Contact( "DB22_DisplayData".dbx20_7 )
   END_RUNG wire#w2
   RUNG wire#powerrail
      Contact( "DB22_DisplayData".dbx20_7 )
      I_Contact( "V50_5" )
      I_Contact( "E43" )
      I_Contact( "In_Pos5" )
   END_RUNG wire#w2
   RUNG wire#powerrail
      Contact( "A34" )
      Contact( "E43" )
   END_RUNG wire#w2
   // the same network as SCL:
   "DB10_ExtConveyors".Out_ConvPos5 := ("V50_5" AND ("V15_6" OR "DB22_DisplayData".dbx20_7)) OR ("DB22_DisplayData".dbx20_7 AND NOT "V50_5" AND NOT "E43" AND NOT "In_Pos5") OR ("A34" AND "E43");
END_REGION

REGION Network 23: Pallet ready in infeed signal (Std signal)
   RUNG wire#powerrail
      Contact( "On" )
      wire#w1
      Contact( "Auto" )
      wire#w2
      Contact( "In_Pos5" )
      wire#w3
      S_Coil( "E43" )
   END_RUNG
   RUNG wire#w1
      Contact( "DB22_DisplayData".dbx20_0 )
   END_RUNG wire#w2
   RUNG wire#w3
      Contact( "V51_5" )
      wire#w4
      S_Coil( "E46" )
   END_RUNG
   RUNG wire#w4
      R_Coil( "V51_5" )
   END_RUNG
   RUNG wire#w1
      Contact( "A35" )
      wire#w5
      R_Coil( "E43" )
   END_RUNG
   RUNG wire#w5
      R_Coil( "E46" )
   END_RUNG
   // the same network as SCL:
   #_w1 := "On" AND ("Auto" OR "DB22_DisplayData".dbx20_0) AND "In_Pos5";
   IF #_w1 THEN "E43" := TRUE; END_IF;
   IF #_w1 AND "V51_5" THEN
       "E46" := TRUE;
       "V51_5" := FALSE;
   END_IF;
   IF "On" AND "A35" THEN
       "E43" := FALSE;
       "E46" := FALSE;
   END_IF;
END_REGION

REGION Network 24: Memory to exclude wrapping in pos 1
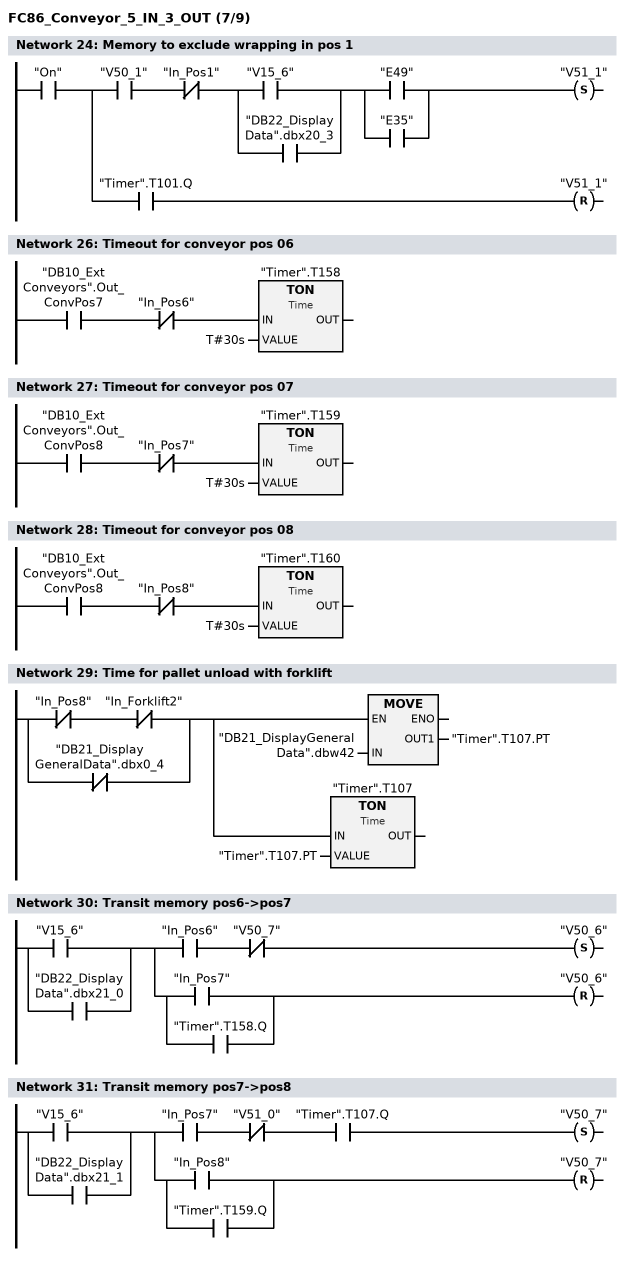
   RUNG wire#powerrail
      Contact( "On" )
      wire#w1
      Contact( "V50_1" )
      I_Contact( "In_Pos1" )
      wire#w2
      Contact( "V15_6" )
      wire#w3
      Contact( "E49" )
      wire#w4
      S_Coil( "V51_1" )
   END_RUNG
   RUNG wire#w2
      Contact( "DB22_DisplayData".dbx20_3 )
   END_RUNG wire#w3
   RUNG wire#w3
      Contact( "E35" )
   END_RUNG wire#w4
   RUNG wire#w1
      Contact( "Timer".T101.Q )
      R_Coil( "V51_1" )
   END_RUNG
   // the same network as SCL:
   IF "On" AND "V50_1" AND NOT "In_Pos1" AND ("V15_6" OR "DB22_DisplayData".dbx20_3) AND ("E49" OR "E35") THEN
       "V51_1" := TRUE;
   END_IF;
   IF "On" AND "Timer".T101.Q THEN "V51_1" := FALSE; END_IF;
END_REGION

REGION Network 25: >>>>>>> OUTFEED CONVEYOR <<<<<<<<
END_REGION

REGION Network 26: Timeout for conveyor pos 06
   "Timer".T158.TON(IN := "DB10_ExtConveyors".Out_ConvPos7 AND NOT "In_Pos6", PT := T#30s);   // TON coil
END_REGION

REGION Network 27: Timeout for conveyor pos 07
   "Timer".T159.TON(IN := "DB10_ExtConveyors".Out_ConvPos8 AND NOT "In_Pos7", PT := T#30s);   // TON coil
END_REGION

REGION Network 28: Timeout for conveyor pos 08
   "Timer".T160.TON(IN := "DB10_ExtConveyors".Out_ConvPos8 AND NOT "In_Pos8", PT := T#30s);   // TON coil
END_REGION

REGION Network 29: Time for pallet unload with forklift
   #_w1 := (NOT "In_Pos8" AND NOT "In_Forklift2") OR NOT "DB21_DisplayGeneralData".dbx0_4;
   IF #_w1 THEN "Timer".T107.PT := "DB21_DisplayGeneralData".dbw42; END_IF;
   "Timer".T107.TON(IN := #_w1, PT := "Timer".T107.PT);   // TON coil
END_REGION

REGION Network 30: Transit memory pos6->pos7
   RUNG wire#powerrail
      Contact( "V15_6" )
      wire#w1
      Contact( "In_Pos6" )
      I_Contact( "V50_7" )
      S_Coil( "V50_6" )
   END_RUNG
   RUNG wire#powerrail
      Contact( "DB22_DisplayData".dbx21_0 )
   END_RUNG wire#w1
   RUNG wire#w1
      Contact( "In_Pos7" )
      wire#w2
      R_Coil( "V50_6" )
   END_RUNG
   RUNG wire#w1
      Contact( "Timer".T158.Q )
   END_RUNG wire#w2
   // the same network as SCL:
   #_w1 := "V15_6" OR "DB22_DisplayData".dbx21_0;
   IF #_w1 AND "In_Pos6" AND NOT "V50_7" THEN "V50_6" := TRUE; END_IF;
   IF #_w1 AND ("In_Pos7" OR "Timer".T158.Q) THEN "V50_6" := FALSE; END_IF;
END_REGION

REGION Network 31: Transit memory pos7->pos8
   RUNG wire#powerrail
      Contact( "V15_6" )
      wire#w1
      Contact( "In_Pos7" )
      I_Contact( "V51_0" )
      Contact( "Timer".T107.Q )
      S_Coil( "V50_7" )
   END_RUNG
   RUNG wire#powerrail
      Contact( "DB22_DisplayData".dbx21_1 )
   END_RUNG wire#w1
   RUNG wire#w1
      Contact( "In_Pos8" )
      wire#w2
      R_Coil( "V50_7" )
   END_RUNG
   RUNG wire#w1
      Contact( "Timer".T159.Q )
   END_RUNG wire#w2
   // the same network as SCL:
   #_w1 := "V15_6" OR "DB22_DisplayData".dbx21_1;
   IF #_w1 AND "In_Pos7" AND NOT "V51_0" AND "Timer".T107.Q THEN "V50_7" := TRUE; END_IF;
   IF #_w1 AND ("In_Pos8" OR "Timer".T159.Q) THEN "V50_7" := FALSE; END_IF;
END_REGION

REGION Network 32: Outfeed conveyor pos.8 unload
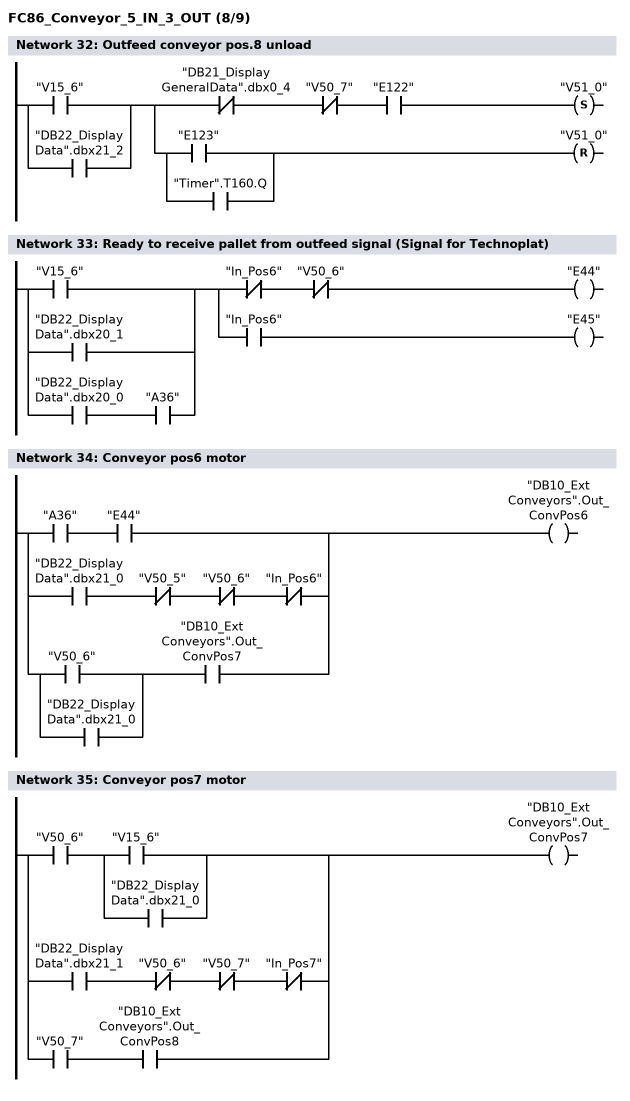
   RUNG wire#powerrail
      Contact( "V15_6" )
      wire#w1
      I_Contact( "DB21_DisplayGeneralData".dbx0_4 )
      I_Contact( "V50_7" )
      Contact( "E122" )
      S_Coil( "V51_0" )
   END_RUNG
   RUNG wire#powerrail
      Contact( "DB22_DisplayData".dbx21_2 )
   END_RUNG wire#w1
   RUNG wire#w1
      Contact( "E123" )
      wire#w2
      R_Coil( "V51_0" )
   END_RUNG
   RUNG wire#w1
      Contact( "Timer".T160.Q )
   END_RUNG wire#w2
   // the same network as SCL:
   #_w1 := "V15_6" OR "DB22_DisplayData".dbx21_2;
   IF #_w1 AND NOT "DB21_DisplayGeneralData".dbx0_4 AND NOT "V50_7" AND "E122" THEN "V51_0" := TRUE; END_IF;
   IF #_w1 AND ("E123" OR "Timer".T160.Q) THEN "V51_0" := FALSE; END_IF;
END_REGION

REGION Network 33: Ready to receive pallet from outfeed signal (Signal for Technoplat)
   RUNG wire#powerrail
      Contact( "V15_6" )
      wire#w1
      I_Contact( "In_Pos6" )
      I_Contact( "V50_6" )
      Coil( "E44" )
   END_RUNG
   RUNG wire#powerrail
      Contact( "DB22_DisplayData".dbx20_1 )
   END_RUNG wire#w1
   RUNG wire#powerrail
      Contact( "DB22_DisplayData".dbx20_0 )
      Contact( "A36" )
   END_RUNG wire#w1
   RUNG wire#w1
      Contact( "In_Pos6" )
      Coil( "E45" )
   END_RUNG
   // the same network as SCL:
   #_w1 := "V15_6" OR "DB22_DisplayData".dbx20_1 OR ("DB22_DisplayData".dbx20_0 AND "A36");
   "E44" := #_w1 AND NOT "In_Pos6" AND NOT "V50_6";
   "E45" := #_w1 AND "In_Pos6";
END_REGION

REGION Network 34: Conveyor pos6 motor
   RUNG wire#powerrail
      Contact( "A36" )
      Contact( "E44" )
      wire#w1
      Coil( "DB10_ExtConveyors".Out_ConvPos6 )
   END_RUNG
   RUNG wire#powerrail
      Contact( "DB22_DisplayData".dbx21_0 )
      I_Contact( "V50_5" )
      I_Contact( "V50_6" )
      I_Contact( "In_Pos6" )
   END_RUNG wire#w1
   RUNG wire#powerrail
      Contact( "V50_6" )
      wire#w2
      Contact( "DB10_ExtConveyors".Out_ConvPos7 )
   END_RUNG wire#w1
   RUNG wire#powerrail
      Contact( "DB22_DisplayData".dbx21_0 )
   END_RUNG wire#w2
   // the same network as SCL:
   "DB10_ExtConveyors".Out_ConvPos6 := ("A36" AND "E44") OR ("DB22_DisplayData".dbx21_0 AND NOT "V50_5" AND NOT "V50_6" AND NOT "In_Pos6") OR (("V50_6" OR "DB22_DisplayData".dbx21_0) AND "DB10_ExtConveyors".Out_ConvPos7);
END_REGION

REGION Network 35: Conveyor pos7 motor
   RUNG wire#powerrail
      Contact( "V50_6" )
      wire#w1
      Contact( "V15_6" )
      wire#w2
      Coil( "DB10_ExtConveyors".Out_ConvPos7 )
   END_RUNG
   RUNG wire#w1
      Contact( "DB22_DisplayData".dbx21_0 )
   END_RUNG wire#w2
   RUNG wire#powerrail
      Contact( "DB22_DisplayData".dbx21_1 )
      I_Contact( "V50_6" )
      I_Contact( "V50_7" )
      I_Contact( "In_Pos7" )
   END_RUNG wire#w2
   RUNG wire#powerrail
      Contact( "V50_7" )
      Contact( "DB10_ExtConveyors".Out_ConvPos8 )
   END_RUNG wire#w2
   // the same network as SCL:
   "DB10_ExtConveyors".Out_ConvPos7 := ("V50_6" AND ("V15_6" OR "DB22_DisplayData".dbx21_0)) OR ("DB22_DisplayData".dbx21_1 AND NOT "V50_6" AND NOT "V50_7" AND NOT "In_Pos7") OR ("V50_7" AND "DB10_ExtConveyors".Out_ConvPos8);
END_REGION

REGION Network 36: Conveyor pos8 motor
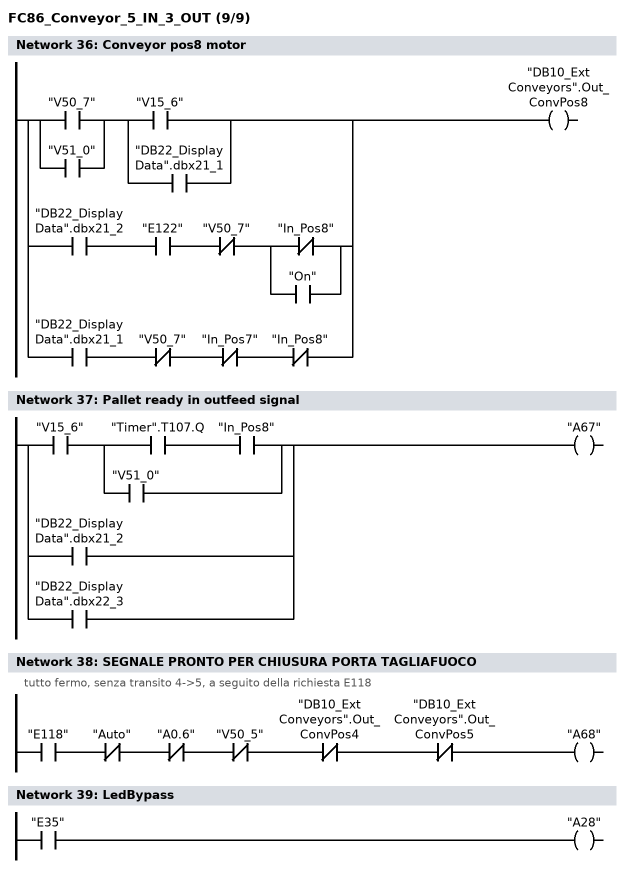
   RUNG wire#powerrail
      Contact( "V50_7" )
      wire#w1
      Contact( "V15_6" )
      wire#w2
      Coil( "DB10_ExtConveyors".Out_ConvPos8 )
   END_RUNG
   RUNG wire#powerrail
      Contact( "V51_0" )
   END_RUNG wire#w1
   RUNG wire#w1
      Contact( "DB22_DisplayData".dbx21_1 )
   END_RUNG wire#w2
   RUNG wire#powerrail
      Contact( "DB22_DisplayData".dbx21_2 )
      Contact( "E122" )
      I_Contact( "V50_7" )
      wire#w3
      I_Contact( "In_Pos8" )
   END_RUNG wire#w2
   RUNG wire#w3
      Contact( "On" )
   END_RUNG wire#w2
   RUNG wire#powerrail
      Contact( "DB22_DisplayData".dbx21_1 )
      I_Contact( "V50_7" )
      I_Contact( "In_Pos7" )
      I_Contact( "In_Pos8" )
   END_RUNG wire#w2
   // the same network as SCL:
   "DB10_ExtConveyors".Out_ConvPos8 := (("V50_7" OR "V51_0") AND ("V15_6" OR "DB22_DisplayData".dbx21_1)) OR ("DB22_DisplayData".dbx21_2 AND "E122" AND NOT "V50_7" AND (NOT "In_Pos8" OR "On")) OR ("DB22_DisplayData".dbx21_1 AND NOT "V50_7" AND NOT "In_Pos7" AND NOT "In_Pos8");
END_REGION

REGION Network 37: Pallet ready in outfeed signal
   RUNG wire#powerrail
      Contact( "V15_6" )
      wire#w1
      Contact( "Timer".T107.Q )
      Contact( "In_Pos8" )
      wire#w2
      Coil( "A67" )
   END_RUNG
   RUNG wire#w1
      Contact( "V51_0" )
   END_RUNG wire#w2
   RUNG wire#powerrail
      Contact( "DB22_DisplayData".dbx21_2 )
   END_RUNG wire#w2
   RUNG wire#powerrail
      Contact( "DB22_DisplayData".dbx22_3 )
   END_RUNG wire#w2
   // the same network as SCL:
   "A67" := ("V15_6" AND (("Timer".T107.Q AND "In_Pos8") OR "V51_0")) OR "DB22_DisplayData".dbx21_2 OR "DB22_DisplayData".dbx22_3;
END_REGION

REGION Network 38: SEGNALE PRONTO PER CHIUSURA PORTA TAGLIAFUOCO
   // tutto fermo, senza transito 4->5, a seguito della richiesta E118
   RUNG wire#powerrail
      Contact( "E118" )
      I_Contact( "Auto" )
      I_Contact( "A0.6" )
      I_Contact( "V50_5" )
      I_Contact( "DB10_ExtConveyors".Out_ConvPos4 )
      I_Contact( "DB10_ExtConveyors".Out_ConvPos5 )
      Coil( "A68" )
   END_RUNG
   // the same network as SCL:
   "A68" := "E118" AND NOT "Auto" AND NOT "A0.6" AND NOT "V50_5" AND NOT "DB10_ExtConveyors".Out_ConvPos4 AND NOT "DB10_ExtConveyors".Out_ConvPos5;
END_REGION

REGION Network 39: LedBypass
   RUNG wire#powerrail
      Contact( "E35" )
      Coil( "A28" )
   END_RUNG
   // the same network as SCL:
   "A28" := "E35";
END_REGION
END_FUNCTION

FUNCTION "Inverter_CW_Assembly" : Void   // FC16, FBD
{ S7_Optimized_Access := 'TRUE' }
VERSION : 0.1
// stored: AutoNumber false, IsIECCheckEnabled false, SetENOAutomatically false, UDAEnableTagReadback false
   VAR_INPUT
      CW_Off1_On : Bool;
      CW_Off2 : Bool;
      CW_Off3 : Bool;
      CW_enable_operation : Bool;
      CW_no_lock_RFG : Bool;
      CW_no_stop_RFG : Bool;
      CW_enable_setpoint : Bool;
      CW_acknowledge : Bool;
      CW_not_used_1 : Bool;
      CW_not_used_2 : Bool;
      CW_PLC_is_Master : Bool;
      CW_direction_reversal : Bool;
      CW_not_used_3 : Bool;
      CW_motortpoti_up : Bool;
      CW_motortpoti_down : Bool;
      CW_not_used_4 : Bool;
   END_VAR
   VAR_IN_OUT
      Control_word : Word;
   END_VAR
BEGIN

REGION Network 1
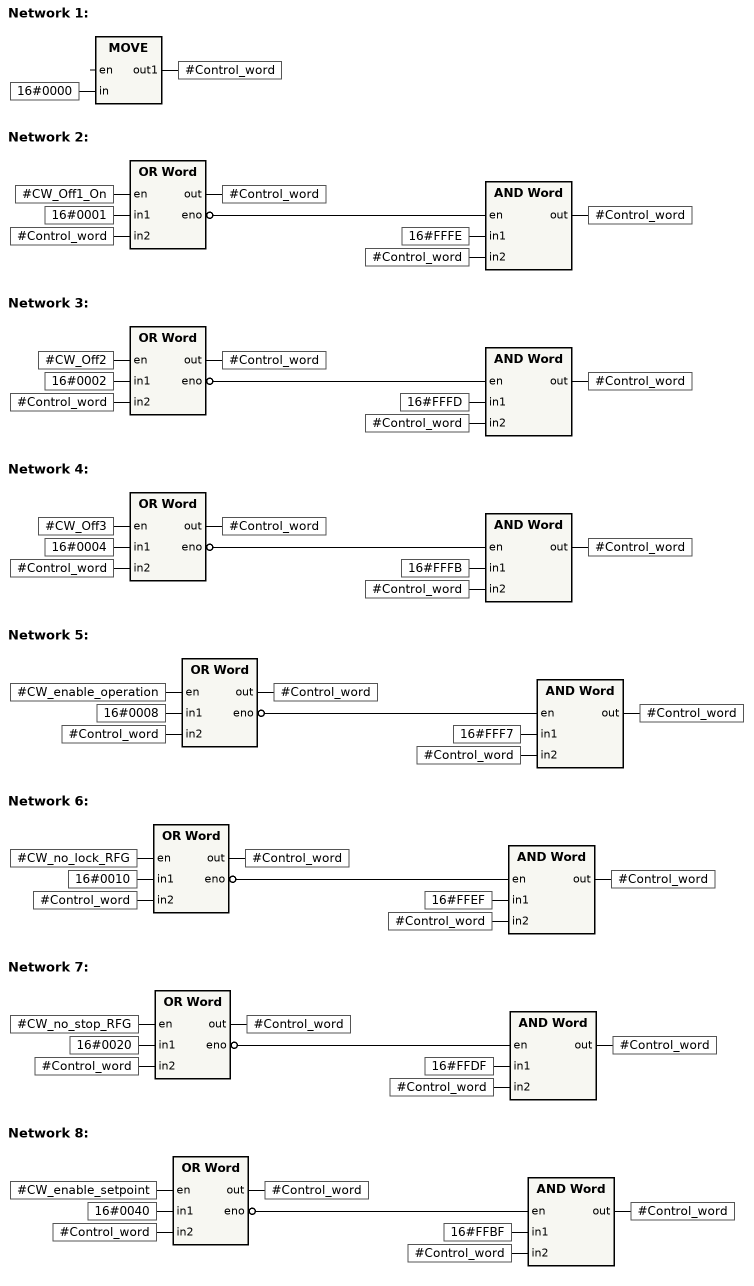
   #Control_word := 16#0000;
END_REGION

REGION Network 2
   IF #CW_Off1_On THEN #Control_word := 16#0001 OR #Control_word; END_IF;
   IF NOT #CW_Off1_On THEN #Control_word := 16#FFFE AND #Control_word; END_IF;
END_REGION

REGION Network 3
   IF #CW_Off2 THEN #Control_word := 16#0002 OR #Control_word; END_IF;
   IF NOT #CW_Off2 THEN #Control_word := 16#FFFD AND #Control_word; END_IF;
END_REGION

REGION Network 4
   IF #CW_Off3 THEN #Control_word := 16#0004 OR #Control_word; END_IF;
   IF NOT #CW_Off3 THEN #Control_word := 16#FFFB AND #Control_word; END_IF;
END_REGION

REGION Network 5
   IF #CW_enable_operation THEN #Control_word := 16#0008 OR #Control_word; END_IF;
   IF NOT #CW_enable_operation THEN #Control_word := 16#FFF7 AND #Control_word; END_IF;
END_REGION

REGION Network 6
   IF #CW_no_lock_RFG THEN #Control_word := 16#0010 OR #Control_word; END_IF;
   IF NOT #CW_no_lock_RFG THEN #Control_word := 16#FFEF AND #Control_word; END_IF;
END_REGION

REGION Network 7
   IF #CW_no_stop_RFG THEN #Control_word := 16#0020 OR #Control_word; END_IF;
   IF NOT #CW_no_stop_RFG THEN #Control_word := 16#FFDF AND #Control_word; END_IF;
END_REGION

REGION Network 8
   IF #CW_enable_setpoint THEN #Control_word := 16#0040 OR #Control_word; END_IF;
   IF NOT #CW_enable_setpoint THEN #Control_word := 16#FFBF AND #Control_word; END_IF;
END_REGION

REGION Network 9
